Yaskawa INFORM job: DEMO_ROOF_UPPER_0625_3PAINT_49.JBI

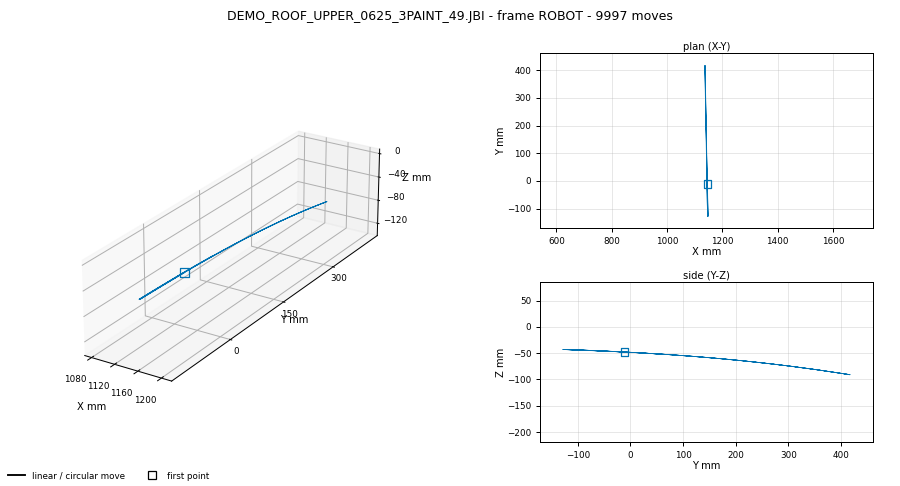
[picture p0: tool path of DEMO_ROOF_UPPER_0625_3PAINT_49.JBI in frame ROBOT, 9997 of 9997 moves have a stored position in this frame; points joined in program order, loops and branches not executed]
/JOB
//NAME DEMO_ROOF_UPPER_0625_3PAINT49
//POS
///NPOS 9997,0,0,0,0,0
///TOOL 0
///USER 0
///POSTYPE ROBOT
///RECTAN
///RCONF 1,0,0,0,0,0,0,0,0,0,0,0,0,0,0,0,0,0,0,0,0,0,0,0
C00000=1146.080,-11.263,-47.724,179.579,6.166,149.236
C00001=1146.085,-11.512,-47.711,179.577,6.165,149.237
C00002=1146.092,-11.763,-47.699,179.574,6.165,149.238
C00003=1146.097,-12.012,-47.686,179.572,6.164,149.238
C00004=1146.101,-12.262,-47.673,179.570,6.163,149.239
C00005=1146.106,-12.511,-47.661,179.567,6.163,149.239
C00006=1146.112,-12.761,-47.648,179.565,6.162,149.240
C00007=1146.117,-13.010,-47.635,179.563,6.161,149.240
C00008=1146.122,-13.261,-47.623,179.560,6.161,149.241
C00009=1146.127,-13.510,-47.610,179.558,6.160,149.242
C00010=1146.132,-13.760,-47.597,179.555,6.159,149.242
C00011=1146.138,-14.009,-47.585,179.552,6.158,149.243
C00012=1146.143,-14.258,-47.572,179.550,6.157,149.243
C00013=1146.148,-14.509,-47.560,179.548,6.156,149.244
C00014=1146.153,-14.758,-47.547,179.545,6.156,149.244
C00015=1146.158,-15.007,-47.535,179.543,6.155,149.245
C00016=1146.163,-15.257,-47.522,179.540,6.155,149.245
C00017=1146.169,-15.507,-47.510,179.538,6.154,149.246
C00018=1146.174,-15.756,-47.497,179.536,6.154,149.247
C00019=1146.179,-16.006,-47.484,179.533,6.153,149.247
C00020=1146.184,-16.256,-47.472,179.531,6.152,149.248
C00021=1146.189,-16.506,-47.460,179.529,6.152,149.248
C00022=1146.194,-16.755,-47.447,179.526,6.151,149.249
C00023=1146.200,-17.004,-47.434,179.523,6.150,149.249
C00024=1146.205,-17.254,-47.422,179.521,6.149,149.250
C00025=1146.210,-17.503,-47.410,179.518,6.148,149.251
C00026=1146.215,-17.753,-47.397,179.516,6.148,149.251
C00027=1146.220,-18.003,-47.385,179.514,6.147,149.252
C00028=1146.225,-18.253,-47.372,179.511,6.146,149.252
C00029=1146.231,-18.503,-47.361,179.509,6.146,149.253
C00030=1146.236,-18.752,-47.348,179.506,6.145,149.253
C00031=1146.241,-19.001,-47.335,179.504,6.144,149.254
C00032=1146.246,-19.251,-47.323,179.502,6.144,149.254
C00033=1146.251,-19.501,-47.311,179.499,6.143,149.255
C00034=1146.256,-19.751,-47.299,179.497,6.142,149.256
C00035=1146.261,-20.001,-47.286,179.495,6.142,149.256
C00036=1146.266,-20.250,-47.273,179.492,6.141,149.257
C00037=1146.272,-20.500,-47.262,179.490,6.141,149.257
C00038=1146.277,-20.749,-47.249,179.488,6.140,149.258
C00039=1146.282,-20.999,-47.237,179.485,6.139,149.258
C00040=1146.288,-21.248,-47.224,179.483,6.139,149.259
C00041=1146.293,-21.498,-47.213,179.481,6.138,149.259
C00042=1146.298,-21.748,-47.200,179.477,6.137,149.260
C00043=1146.304,-21.998,-47.188,179.475,6.136,149.261
C00044=1146.309,-22.247,-47.175,179.472,6.135,149.261
C00045=1146.314,-22.497,-47.164,179.470,6.135,149.262
C00046=1146.319,-22.746,-47.151,179.468,6.134,149.262
C00047=1146.325,-22.996,-47.139,179.465,6.133,149.263
C00048=1146.330,-23.245,-47.127,179.463,6.133,149.263
C00049=1146.335,-23.496,-47.114,179.461,6.132,149.264
C00050=1146.340,-23.745,-47.102,179.458,6.131,149.265
C00051=1146.345,-23.995,-47.090,179.456,6.131,149.265
C00052=1146.351,-24.264,-47.076,179.454,6.130,149.266
C00053=1146.356,-24.535,-47.063,179.451,6.130,149.266
C00054=1146.361,-24.805,-47.051,179.449,6.129,149.267
C00055=1146.367,-25.075,-47.038,179.445,6.128,149.268
C00056=1146.372,-25.324,-47.025,179.443,6.127,149.268
C00057=1146.378,-25.574,-47.013,179.441,6.127,149.269
C00058=1146.383,-25.824,-47.002,179.438,6.126,149.269
C00059=1146.388,-26.073,-46.989,179.436,6.125,149.270
C00060=1146.394,-26.323,-46.977,179.434,6.125,149.270
C00061=1146.399,-26.572,-46.964,179.431,6.124,149.271
C00062=1146.404,-26.822,-46.953,179.429,6.123,149.272
C00063=1146.409,-27.072,-46.941,179.427,6.123,149.272
C00064=1146.414,-27.321,-46.929,179.424,6.122,149.273
C00065=1146.420,-27.571,-46.917,179.422,6.121,149.273
C00066=1146.425,-27.821,-46.905,179.419,6.121,149.274
C00067=1146.429,-28.070,-46.893,179.417,6.120,149.274
C00068=1146.435,-28.320,-46.881,179.415,6.119,149.275
C00069=1146.440,-28.570,-46.869,179.412,6.119,149.276
C00070=1146.445,-28.819,-46.857,179.410,6.118,149.276
C00071=1146.451,-29.069,-46.845,179.407,6.118,149.277
C00072=1146.456,-29.319,-46.833,179.405,6.117,149.277
C00073=1146.461,-29.568,-46.821,179.402,6.117,149.278
C00074=1146.466,-29.818,-46.809,179.400,6.116,149.278
C00075=1146.472,-30.068,-46.797,179.398,6.115,149.279
C00076=1146.476,-30.318,-46.786,179.395,6.115,149.280
C00077=1146.481,-30.567,-46.773,179.393,6.114,149.280
C00078=1146.487,-30.817,-46.761,179.390,6.113,149.281
C00079=1146.492,-31.067,-46.749,179.388,6.113,149.281
C00080=1146.497,-31.317,-46.738,179.387,6.113,149.282
C00081=1146.503,-31.566,-46.727,179.384,6.112,149.282
C00082=1146.508,-31.815,-46.714,179.382,6.111,149.283
C00083=1146.513,-32.065,-46.702,179.379,6.111,149.284
C00084=1146.518,-32.315,-46.691,179.377,6.110,149.284
C00085=1146.524,-32.565,-46.679,179.374,6.110,149.285
C00086=1146.529,-32.815,-46.667,179.372,6.109,149.285
C00087=1146.533,-33.064,-46.655,179.370,6.108,149.286
C00088=1146.539,-33.313,-46.643,179.367,6.108,149.286
C00089=1146.544,-33.563,-46.631,179.365,6.107,149.287
C00090=1146.549,-33.813,-46.620,179.362,6.107,149.288
C00091=1146.555,-34.062,-46.608,179.360,6.106,149.288
C00092=1146.560,-34.312,-46.597,179.358,6.105,149.289
C00093=1146.565,-34.562,-46.585,179.355,6.105,149.289
C00094=1146.570,-34.811,-46.573,179.353,6.104,149.290
C00095=1146.576,-35.061,-46.561,179.351,6.103,149.290
C00096=1146.580,-35.311,-46.549,179.348,6.103,149.291
C00097=1146.586,-35.561,-46.538,179.346,6.102,149.291
C00098=1146.592,-35.810,-46.526,179.344,6.101,149.292
C00099=1146.596,-36.060,-46.515,179.341,6.101,149.293
C00100=1146.602,-36.309,-46.503,179.339,6.100,149.293
C00101=1146.607,-36.559,-46.492,179.336,6.099,149.294
C00102=1146.612,-36.809,-46.480,179.334,6.099,149.294
C00103=1146.617,-37.059,-46.468,179.332,6.098,149.295
C00104=1146.622,-37.309,-46.457,179.329,6.097,149.295
C00105=1146.628,-37.558,-46.445,179.327,6.097,149.296
C00106=1146.633,-37.807,-46.434,179.325,6.097,149.297
C00107=1146.638,-38.057,-46.422,179.323,6.097,149.297
C00108=1146.644,-38.307,-46.410,179.320,6.096,149.298
C00109=1146.648,-38.557,-46.399,179.318,6.095,149.298
C00110=1146.654,-38.806,-46.387,179.315,6.095,149.299
C00111=1146.659,-39.056,-46.376,179.313,6.094,149.299
C00112=1146.665,-39.306,-46.364,179.311,6.093,149.300
C00113=1146.670,-39.556,-46.352,179.308,6.093,149.301
C00114=1146.675,-39.805,-46.341,179.306,6.092,149.301
C00115=1146.681,-40.055,-46.329,179.304,6.091,149.302
C00116=1146.685,-40.304,-46.318,179.301,6.091,149.302
C00117=1146.691,-40.554,-46.306,179.299,6.090,149.303
C00118=1146.696,-40.804,-46.295,179.297,6.089,149.303
C00119=1146.701,-41.054,-46.283,179.294,6.089,149.304
C00120=1146.706,-41.303,-46.272,179.292,6.088,149.305
C00121=1146.712,-41.553,-46.260,179.290,6.088,149.305
C00122=1146.717,-41.803,-46.250,179.287,6.088,149.306
C00123=1146.722,-42.053,-46.238,179.285,6.087,149.306
C00124=1146.727,-42.302,-46.227,179.283,6.086,149.307
C00125=1146.733,-42.552,-46.215,179.280,6.086,149.307
C00126=1146.738,-42.801,-46.204,179.278,6.085,149.308
C00127=1146.743,-43.051,-46.192,179.276,6.084,149.308
C00128=1146.748,-43.300,-46.181,179.273,6.084,149.309
C00129=1146.754,-43.551,-46.170,179.271,6.083,149.310
C00130=1146.759,-43.800,-46.158,179.269,6.083,149.310
C00131=1146.763,-44.050,-46.147,179.266,6.082,149.311
C00132=1146.769,-44.299,-46.135,179.264,6.081,149.311
C00133=1146.774,-44.549,-46.124,179.262,6.082,149.312
C00134=1146.780,-44.799,-46.112,179.260,6.081,149.312
C00135=1146.785,-45.049,-46.102,179.257,6.080,149.313
C00136=1146.791,-45.298,-46.090,179.255,6.080,149.314
C00137=1146.795,-45.548,-46.079,179.253,6.079,149.314
C00138=1146.800,-45.797,-46.068,179.250,6.078,149.315
C00139=1146.806,-46.047,-46.057,179.248,6.078,149.315
C00140=1146.811,-46.297,-46.046,179.245,6.077,149.316
C00141=1146.816,-46.547,-46.034,179.243,6.076,149.316
C00142=1146.822,-46.796,-46.023,179.242,6.076,149.317
C00143=1146.827,-47.046,-46.012,179.239,6.076,149.318
C00144=1146.832,-47.296,-46.000,179.237,6.075,149.318
C00145=1146.837,-47.545,-45.989,179.234,6.075,149.319
C00146=1146.843,-47.795,-45.977,179.232,6.074,149.319
C00147=1146.848,-48.045,-45.967,179.230,6.073,149.320
C00148=1146.853,-48.294,-45.956,179.227,6.073,149.320
C00149=1146.859,-48.544,-45.944,179.225,6.072,149.321
C00150=1146.864,-48.794,-45.933,179.223,6.071,149.321
C00151=1146.869,-49.043,-45.923,179.221,6.072,149.322
C00152=1146.874,-49.293,-45.911,179.218,6.071,149.322
C00153=1146.879,-49.543,-45.900,179.216,6.071,149.323
C00154=1146.885,-49.792,-45.889,179.214,6.070,149.324
C00155=1146.890,-50.042,-45.877,179.211,6.069,149.324
C00156=1146.895,-50.313,-45.866,179.209,6.069,149.325
C00157=1146.901,-50.583,-45.854,179.206,6.068,149.326
C00158=1146.907,-50.854,-45.841,179.204,6.067,149.326
C00159=1146.912,-51.125,-45.829,179.201,6.067,149.327
C00160=1146.918,-51.375,-45.819,179.199,6.066,149.327
C00161=1146.923,-51.624,-45.808,179.197,6.065,149.328
C00162=1146.929,-51.874,-45.797,179.194,6.065,149.328
C00163=1146.934,-52.124,-45.786,179.192,6.064,149.329
C00164=1146.938,-52.373,-45.774,179.190,6.065,149.330
C00165=1146.945,-52.623,-45.764,179.188,6.064,149.330
C00166=1146.949,-52.873,-45.752,179.185,6.063,149.331
C00167=1146.954,-53.123,-45.742,179.183,6.063,149.331
C00168=1146.960,-53.372,-45.731,179.181,6.062,149.332
C00169=1146.965,-53.622,-45.720,179.178,6.061,149.332
C00170=1146.971,-53.871,-45.709,179.176,6.061,149.333
C00171=1146.976,-54.122,-45.698,179.174,6.061,149.333
C00172=1146.981,-54.371,-45.687,179.171,6.060,149.334
C00173=1146.986,-54.621,-45.677,179.169,6.060,149.335
C00174=1146.991,-54.871,-45.665,179.167,6.059,149.335
C00175=1146.997,-55.120,-45.655,179.164,6.058,149.336
C00176=1147.002,-55.370,-45.643,179.162,6.058,149.336
C00177=1147.007,-55.619,-45.633,179.161,6.058,149.337
C00178=1147.012,-55.869,-45.622,179.158,6.057,149.337
C00179=1147.018,-56.120,-45.611,179.156,6.057,149.338
C00180=1147.023,-56.369,-45.600,179.154,6.056,149.338
C00181=1147.028,-56.619,-45.589,179.151,6.055,149.339
C00182=1147.033,-56.868,-45.578,179.149,6.055,149.340
C00183=1147.038,-57.118,-45.568,179.146,6.054,149.340
C00184=1147.044,-57.368,-45.557,179.144,6.054,149.341
C00185=1147.049,-57.617,-45.546,179.142,6.053,149.341
C00186=1147.055,-57.867,-45.535,179.140,6.053,149.342
C00187=1147.060,-58.117,-45.524,179.137,6.052,149.342
C00188=1147.065,-58.366,-45.514,179.135,6.051,149.343
C00189=1147.070,-58.616,-45.503,179.133,6.052,149.344
C00190=1147.076,-58.865,-45.492,179.131,6.051,149.344
C00191=1147.081,-59.116,-45.482,179.129,6.050,149.345
C00192=1147.085,-59.365,-45.470,179.126,6.050,149.345
C00193=1147.091,-59.615,-45.460,179.124,6.049,149.346
C00194=1147.097,-59.865,-45.449,179.121,6.049,149.346
C00195=1147.102,-60.114,-45.438,179.120,6.049,149.347
C00196=1147.107,-60.364,-45.428,179.118,6.048,149.347
C00197=1147.112,-60.614,-45.417,179.115,6.048,149.348
C00198=1147.117,-60.864,-45.406,179.113,6.047,149.349
C00199=1147.123,-61.113,-45.396,179.110,6.046,149.349
C00200=1147.128,-61.363,-45.385,179.108,6.046,149.350
C00201=1147.133,-61.613,-45.375,179.106,6.046,149.350
C00202=1147.139,-61.862,-45.364,179.104,6.045,149.351
C00203=1147.144,-62.112,-45.354,179.101,6.045,149.351
C00204=1147.149,-62.362,-45.343,179.099,6.044,149.352
C00205=1147.154,-62.611,-45.332,179.097,6.043,149.352
C00206=1147.159,-62.861,-45.322,179.095,6.043,149.353
C00207=1147.164,-63.111,-45.311,179.093,6.043,149.354
C00208=1147.170,-63.361,-45.301,179.091,6.042,149.354
C00209=1147.175,-63.610,-45.290,179.088,6.041,149.355
C00210=1147.180,-63.860,-45.280,179.086,6.041,149.355
C00211=1147.186,-64.110,-45.268,179.084,6.041,149.356
C00212=1147.192,-64.360,-45.258,179.081,6.040,149.356
C00213=1147.197,-64.610,-45.248,179.079,6.040,149.357
C00214=1147.202,-64.859,-45.237,179.077,6.039,149.358
C00215=1147.208,-65.109,-45.226,179.074,6.038,149.358
C00216=1147.213,-65.359,-45.216,179.073,6.038,149.359
C00217=1147.218,-65.608,-45.206,179.070,6.038,149.359
C00218=1147.222,-65.858,-45.196,179.068,6.037,149.360
C00219=1147.228,-66.107,-45.185,179.066,6.036,149.360
C00220=1147.233,-66.357,-45.175,179.064,6.037,149.361
C00221=1147.238,-66.607,-45.164,179.061,6.036,149.361
C00222=1147.244,-66.857,-45.154,179.059,6.035,149.362
C00223=1147.249,-67.107,-45.143,179.057,6.035,149.363
C00224=1147.255,-67.356,-45.133,179.054,6.034,149.363
C00225=1147.260,-67.606,-45.123,179.053,6.034,149.364
C00226=1147.265,-67.856,-45.111,179.050,6.034,149.364
C00227=1147.270,-68.105,-45.101,179.048,6.033,149.365
C00228=1147.275,-68.355,-45.091,179.046,6.032,149.365
C00229=1147.281,-68.605,-45.080,179.044,6.033,149.366
C00230=1147.287,-68.854,-45.070,179.041,6.032,149.366
C00231=1147.292,-69.105,-45.060,179.039,6.031,149.367
C00232=1147.297,-69.354,-45.049,179.037,6.031,149.368
C00233=1147.303,-69.604,-45.039,179.034,6.030,149.368
C00234=1147.308,-69.854,-45.029,179.033,6.030,149.369
C00235=1147.313,-70.103,-45.019,179.030,6.030,149.369
C00236=1147.318,-70.353,-45.009,179.028,6.029,149.370
C00237=1147.323,-70.603,-44.998,179.026,6.028,149.370
C00238=1147.329,-70.853,-44.988,179.024,6.028,149.371
C00239=1147.334,-71.103,-44.978,179.022,6.028,149.371
C00240=1147.339,-71.352,-44.967,179.019,6.027,149.372
C00241=1147.345,-71.602,-44.957,179.017,6.026,149.372
C00242=1147.350,-71.852,-44.947,179.015,6.027,149.373
C00243=1147.355,-72.101,-44.937,179.013,6.026,149.374
C00244=1147.361,-72.351,-44.927,179.011,6.025,149.374
C00245=1147.366,-72.601,-44.916,179.008,6.025,149.375
C00246=1147.371,-72.851,-44.906,179.006,6.025,149.375
C00247=1147.377,-73.100,-44.896,179.004,6.024,149.376
C00248=1147.382,-73.350,-44.886,179.002,6.024,149.376
C00249=1147.387,-73.600,-44.875,178.999,6.023,149.377
C00250=1147.392,-73.849,-44.865,178.998,6.023,149.377
C00251=1147.398,-74.099,-44.855,178.995,6.022,149.378
C00252=1147.403,-74.349,-44.845,178.993,6.022,149.379
C00253=1147.408,-74.599,-44.834,178.991,6.021,149.379
C00254=1147.414,-74.848,-44.824,178.989,6.021,149.380
C00255=1147.418,-75.098,-44.814,178.986,6.020,149.380
C00256=1147.424,-75.348,-44.804,178.984,6.020,149.381
C00257=1147.429,-75.597,-44.794,178.982,6.019,149.381
C00258=1147.435,-75.847,-44.784,178.980,6.019,149.382
C00259=1147.440,-76.098,-44.774,178.978,6.019,149.382
C00260=1147.446,-76.368,-44.763,178.975,6.018,149.383
C00261=1147.451,-76.639,-44.752,178.973,6.017,149.384
C00262=1147.457,-76.911,-44.741,178.970,6.017,149.384
C00263=1147.463,-77.182,-44.731,178.968,6.016,149.385
C00264=1147.468,-77.433,-44.720,178.966,6.016,149.385
C00265=1147.474,-77.682,-44.710,178.964,6.016,149.386
C00266=1147.480,-77.932,-44.700,178.962,6.015,149.387
C00267=1147.484,-78.181,-44.690,178.959,6.014,149.387
C00268=1147.490,-78.432,-44.680,178.957,6.015,149.388
C00269=1147.495,-78.681,-44.670,178.955,6.014,149.388
C00270=1147.501,-78.931,-44.660,178.953,6.013,149.389
C00271=1147.506,-79.180,-44.650,178.951,6.013,149.389
C00272=1147.511,-79.430,-44.640,178.949,6.013,149.390
C00273=1147.517,-79.680,-44.630,178.946,6.012,149.390
C00274=1147.521,-79.930,-44.621,178.944,6.011,149.391
C00275=1147.527,-80.179,-44.610,178.942,6.012,149.392
C00276=1147.533,-80.429,-44.600,178.940,6.011,149.392
C00277=1147.537,-80.679,-44.591,178.938,6.010,149.392
C00278=1147.543,-80.929,-44.581,178.936,6.011,149.393
C00279=1147.548,-81.178,-44.570,178.934,6.010,149.394
C00280=1147.553,-81.428,-44.561,178.931,6.009,149.394
C00281=1147.559,-81.678,-44.551,178.929,6.008,149.395
C00282=1147.564,-81.928,-44.541,178.927,6.009,149.395
C00283=1147.569,-82.177,-44.531,178.925,6.008,149.396
C00284=1147.575,-82.427,-44.521,178.923,6.007,149.396
C00285=1147.581,-82.677,-44.511,178.921,6.008,149.397
C00286=1147.585,-82.926,-44.502,178.918,6.007,149.398
C00287=1147.590,-83.176,-44.491,178.916,6.006,149.398
C00288=1147.596,-83.427,-44.482,178.914,6.005,149.398
C00289=1147.601,-83.676,-44.472,178.912,6.006,149.399
C00290=1147.607,-83.925,-44.462,178.910,6.005,149.400
C00291=1147.612,-84.175,-44.453,178.908,6.004,149.400
C00292=1147.618,-84.425,-44.443,178.906,6.004,149.401
C00293=1147.623,-84.675,-44.432,178.903,6.004,149.401
C00294=1147.628,-84.925,-44.423,178.901,6.003,149.402
C00295=1147.633,-85.174,-44.413,178.900,6.003,149.402
C00296=1147.638,-85.424,-44.404,178.897,6.003,149.403
C00297=1147.644,-85.674,-44.394,178.895,6.002,149.404
C00298=1147.650,-85.923,-44.384,178.893,6.002,149.404
C00299=1147.655,-86.173,-44.375,178.891,6.001,149.404
C00300=1147.660,-86.423,-44.364,178.888,6.001,149.405
C00301=1147.665,-86.673,-44.356,178.886,6.000,149.406
C00302=1147.671,-86.923,-44.345,178.884,6.000,149.406
C00303=1147.675,-87.172,-44.336,178.882,5.999,149.407
C00304=1147.681,-87.422,-44.326,178.880,5.999,149.407
C00305=1147.686,-87.671,-44.317,178.878,5.999,149.408
C00306=1147.692,-87.922,-44.307,178.876,5.998,149.408
C00307=1147.697,-88.171,-44.297,178.873,5.998,149.409
C00308=1147.702,-88.422,-44.288,178.872,5.998,149.410
C00309=1147.707,-88.671,-44.278,178.869,5.997,149.410
C00310=1147.713,-88.921,-44.269,178.867,5.996,149.410
C00311=1147.718,-89.170,-44.259,178.865,5.997,149.411
C00312=1147.724,-89.421,-44.249,178.863,5.996,149.412
C00313=1147.729,-89.670,-44.240,178.861,5.995,149.412
C00314=1147.735,-89.920,-44.230,178.859,5.995,149.413
C00315=1147.739,-90.169,-44.221,178.856,5.995,149.413
C00316=1147.745,-90.419,-44.211,178.854,5.994,149.414
C00317=1147.750,-90.669,-44.202,178.853,5.994,149.414
C00318=1147.756,-90.919,-44.192,178.850,5.994,149.415
C00319=1147.760,-91.169,-44.182,178.848,5.993,149.416
C00320=1147.766,-91.419,-44.173,178.846,5.993,149.416
C00321=1147.771,-91.668,-44.163,178.844,5.992,149.416
C00322=1147.777,-91.918,-44.154,178.842,5.992,149.417
C00323=1147.782,-92.167,-44.144,178.840,5.992,149.418
C00324=1147.788,-92.418,-44.134,178.837,5.991,149.418
C00325=1147.793,-92.667,-44.125,178.835,5.991,149.419
C00326=1147.798,-92.917,-44.116,178.834,5.991,149.419
C00327=1147.804,-93.167,-44.106,178.831,5.990,149.420
C00328=1147.809,-93.416,-44.097,178.829,5.989,149.420
C00329=1147.815,-93.666,-44.087,178.827,5.989,149.421
C00330=1147.819,-93.915,-44.078,178.825,5.989,149.421
C00331=1147.825,-94.166,-44.068,178.823,5.989,149.422
C00332=1147.830,-94.415,-44.059,178.821,5.988,149.422
C00333=1147.835,-94.665,-44.050,178.819,5.988,149.423
C00334=1147.841,-94.915,-44.040,178.817,5.988,149.423
C00335=1147.846,-95.165,-44.031,178.815,5.987,149.424
C00336=1147.852,-95.414,-44.021,178.812,5.987,149.425
C00337=1147.857,-95.664,-44.012,178.811,5.987,149.425
C00338=1147.862,-95.914,-44.003,178.808,5.986,149.426
C00339=1147.868,-96.164,-43.993,178.806,5.985,149.426
C00340=1147.873,-96.413,-43.984,178.804,5.985,149.427
C00341=1147.878,-96.663,-43.975,178.802,5.985,149.427
C00342=1147.884,-96.913,-43.965,178.800,5.984,149.428
C00343=1147.889,-97.163,-43.956,178.798,5.984,149.428
C00344=1147.895,-97.413,-43.947,178.796,5.983,149.429
C00345=1147.900,-97.662,-43.937,178.794,5.984,149.429
C00346=1147.905,-97.912,-43.928,178.792,5.983,149.430
C00347=1147.911,-98.162,-43.919,178.789,5.982,149.430
C00348=1147.916,-98.412,-43.910,178.788,5.982,149.431
C00349=1147.921,-98.661,-43.900,178.785,5.982,149.432
C00350=1147.927,-98.911,-43.891,178.783,5.981,149.432
C00351=1147.932,-99.161,-43.882,178.781,5.981,149.433
C00352=1147.937,-99.411,-43.873,178.779,5.980,149.433
C00353=1147.943,-99.661,-43.863,178.778,5.980,149.434
C00354=1147.948,-99.910,-43.854,178.775,5.980,149.434
C00355=1147.953,-100.160,-43.845,178.773,5.979,149.435
C00356=1147.958,-100.410,-43.836,178.771,5.979,149.435
C00357=1147.964,-100.660,-43.826,178.769,5.979,149.436
C00358=1147.969,-100.909,-43.817,178.767,5.979,149.436
C00359=1147.974,-101.159,-43.808,178.765,5.978,149.437
C00360=1147.980,-101.409,-43.798,178.762,5.977,149.437
C00361=1147.985,-101.659,-43.790,178.761,5.977,149.438
C00362=1147.991,-101.908,-43.781,178.759,5.977,149.438
C00363=1147.996,-102.158,-43.771,178.756,5.976,149.439
C00364=1148.002,-102.430,-43.762,178.754,5.976,149.440
C00365=1148.008,-102.702,-43.751,178.752,5.976,149.440
C00366=1148.014,-102.975,-43.742,178.749,5.975,149.441
C00367=1148.019,-103.247,-43.731,178.747,5.975,149.441
C00368=1148.024,-103.497,-43.722,178.746,5.975,149.442
C00369=1148.030,-103.747,-43.714,178.743,5.974,149.442
C00370=1148.036,-103.996,-43.704,178.741,5.974,149.443
C00371=1148.041,-104.246,-43.696,178.739,5.973,149.443
C00372=1148.046,-104.495,-43.686,178.737,5.973,149.444
C00373=1148.051,-104.745,-43.677,178.735,5.973,149.444
C00374=1148.056,-104.995,-43.668,178.733,5.972,149.445
C00375=1148.062,-105.245,-43.659,178.731,5.972,149.446
C00376=1148.067,-105.495,-43.650,178.729,5.972,149.446
C00377=1148.073,-105.745,-43.641,178.727,5.971,149.447
C00378=1148.078,-105.995,-43.632,178.725,5.971,149.447
C00379=1148.084,-106.244,-43.623,178.723,5.970,149.448
C00380=1148.089,-106.494,-43.615,178.721,5.970,149.448
C00381=1148.095,-106.744,-43.605,178.719,5.970,149.449
C00382=1148.100,-106.994,-43.596,178.716,5.969,149.449
C00383=1148.105,-107.243,-43.587,178.715,5.969,149.450
C00384=1148.110,-107.493,-43.578,178.713,5.968,149.450
C00385=1148.115,-107.743,-43.569,178.711,5.968,149.451
C00386=1148.120,-107.993,-43.561,178.709,5.968,149.451
C00387=1148.127,-108.243,-43.551,178.707,5.968,149.452
C00388=1148.132,-108.492,-43.542,178.705,5.967,149.452
C00389=1148.137,-108.742,-43.534,178.702,5.967,149.453
C00390=1148.142,-108.992,-43.525,178.701,5.967,149.453
C00391=1148.148,-109.242,-43.516,178.699,5.966,149.454
C00392=1148.153,-109.492,-43.507,178.697,5.966,149.454
C00393=1148.159,-109.741,-43.498,178.694,5.966,149.455
C00394=1148.164,-109.991,-43.489,178.693,5.966,149.456
C00395=1148.169,-110.241,-43.481,178.691,5.965,149.456
C00396=1148.175,-110.491,-43.471,178.688,5.964,149.457
C00397=1148.180,-110.741,-43.462,178.687,5.964,149.457
C00398=1148.185,-110.990,-43.453,178.685,5.963,149.458
C00399=1148.191,-111.240,-43.445,178.683,5.964,149.458
C00400=1148.196,-111.489,-43.436,178.680,5.963,149.459
C00401=1148.201,-111.739,-43.427,178.679,5.963,149.459
C00402=1148.206,-111.989,-43.418,178.677,5.962,149.460
C00403=1148.212,-112.239,-43.409,178.674,5.962,149.460
C00404=1148.217,-112.488,-43.401,178.673,5.962,149.461
C00405=1148.222,-112.738,-43.392,178.671,5.961,149.461
C00406=1148.228,-112.989,-43.384,178.668,5.961,149.462
C00407=1148.233,-113.238,-43.375,178.666,5.961,149.462
C00408=1148.239,-113.487,-43.366,178.665,5.961,149.463
C00409=1148.245,-113.738,-43.357,178.662,5.960,149.463
C00410=1148.250,-113.988,-43.348,178.660,5.959,149.464
C00411=1148.255,-114.237,-43.339,178.659,5.959,149.464
C00412=1148.260,-114.487,-43.330,178.656,5.958,149.465
C00413=1148.266,-114.737,-43.322,178.654,5.959,149.465
C00414=1148.272,-114.987,-43.313,178.652,5.958,149.466
C00415=1148.277,-115.237,-43.304,178.651,5.958,149.466
C00416=1148.282,-115.487,-43.295,178.648,5.957,149.467
C00417=1148.288,-115.736,-43.287,178.647,5.957,149.467
C00418=1148.293,-115.986,-43.278,178.645,5.957,149.468
C00419=1148.298,-116.236,-43.270,178.642,5.956,149.468
C00420=1148.303,-116.486,-43.261,178.640,5.956,149.469
C00421=1148.309,-116.735,-43.252,178.638,5.956,149.470
C00422=1148.314,-116.985,-43.243,178.637,5.956,149.470
C00423=1148.320,-117.235,-43.235,178.634,5.955,149.471
C00424=1148.326,-117.484,-43.227,178.633,5.955,149.471
C00425=1148.331,-117.734,-43.218,178.631,5.954,149.472
C00426=1148.336,-117.984,-43.209,178.629,5.954,149.472
C00427=1148.341,-118.234,-43.200,178.627,5.953,149.473
C00428=1148.347,-118.484,-43.192,178.625,5.954,149.473
C00429=1148.352,-118.733,-43.184,178.623,5.953,149.474
C00430=1148.357,-118.983,-43.175,178.621,5.953,149.474
C00431=1148.362,-119.233,-43.166,178.619,5.952,149.475
C00432=1148.368,-119.483,-43.158,178.617,5.952,149.475
C00433=1148.373,-119.733,-43.149,178.615,5.952,149.476
C00434=1148.378,-119.983,-43.141,178.613,5.951,149.476
C00435=1148.384,-120.232,-43.133,178.611,5.951,149.477
C00436=1148.390,-120.482,-43.124,178.609,5.950,149.477
C00437=1148.395,-120.732,-43.115,178.607,5.951,149.478
C00438=1148.401,-120.981,-43.106,178.605,5.950,149.478
C00439=1148.406,-121.232,-43.098,178.603,5.950,149.479
C00440=1148.411,-121.481,-43.089,178.601,5.949,149.479
C00441=1148.416,-121.730,-43.081,178.599,5.949,149.480
C00442=1148.422,-121.981,-43.073,178.597,5.948,149.480
C00443=1148.427,-122.231,-43.064,178.595,5.948,149.481
C00444=1148.432,-122.480,-43.055,178.593,5.948,149.481
C00445=1148.438,-122.730,-43.048,178.592,5.948,149.482
C00446=1148.443,-122.980,-43.039,178.589,5.947,149.482
C00447=1148.449,-123.229,-43.030,178.588,5.947,149.483
C00448=1148.454,-123.480,-43.022,178.585,5.947,149.483
C00449=1148.459,-123.729,-43.014,178.584,5.947,149.484
C00450=1148.465,-123.979,-43.006,178.581,5.946,149.484
C00451=1148.470,-124.229,-42.997,178.579,5.945,149.485
C00452=1148.475,-124.479,-42.988,178.578,5.945,149.485
C00453=1148.481,-124.728,-42.980,178.575,5.945,149.486
C00454=1148.487,-124.978,-42.971,178.574,5.945,149.486
C00455=1148.492,-125.229,-42.963,178.572,5.944,149.487
C00456=1148.497,-125.478,-42.955,178.570,5.944,149.487
C00457=1148.502,-125.728,-42.946,178.568,5.943,149.488
C00458=1148.508,-125.978,-42.938,178.566,5.943,149.488
C00459=1148.513,-126.227,-42.930,178.564,5.942,149.489
C00460=1148.519,-126.478,-42.921,178.562,5.943,149.490
C00461=1148.524,-126.726,-42.913,178.560,5.942,149.490
C00462=1148.529,-126.977,-42.905,178.558,5.942,149.491
C00463=1148.535,-127.227,-42.896,178.556,5.941,149.491
C00464=1148.541,-127.477,-42.889,178.554,5.941,149.491
C00465=1148.546,-127.726,-42.880,178.552,5.941,149.492
C00466=1148.551,-127.976,-42.872,178.551,5.941,149.492
C00467=1148.556,-128.226,-42.864,178.548,5.940,149.493
C00468=1148.135,-128.237,-42.906,178.545,5.944,149.495
C00469=1148.130,-127.987,-42.915,178.547,5.944,149.494
C00470=1148.124,-127.737,-42.923,178.549,5.945,149.494
C00471=1148.119,-127.488,-42.931,178.551,5.945,149.493
C00472=1148.114,-127.238,-42.939,178.553,5.945,149.493
C00473=1148.108,-126.988,-42.948,178.555,5.945,149.492
C00474=1148.103,-126.738,-42.956,178.557,5.946,149.492
C00475=1148.098,-126.488,-42.965,178.559,5.946,149.491
C00476=1148.092,-126.239,-42.972,178.561,5.947,149.491
C00477=1148.087,-125.989,-42.981,178.562,5.946,149.490
C00478=1148.082,-125.739,-42.990,178.565,5.947,149.490
C00479=1148.076,-125.489,-42.998,178.566,5.947,149.489
C00480=1148.071,-125.239,-43.007,178.568,5.948,149.489
C00481=1148.065,-124.990,-43.014,178.570,5.948,149.488
C00482=1148.060,-124.740,-43.023,178.572,5.949,149.488
C00483=1148.055,-124.490,-43.031,178.574,5.949,149.487
C00484=1148.049,-124.240,-43.039,178.576,5.949,149.487
C00485=1148.044,-123.991,-43.048,178.578,5.949,149.486
C00486=1148.038,-123.740,-43.056,178.580,5.950,149.486
C00487=1148.032,-123.491,-43.065,178.582,5.950,149.485
C00488=1148.028,-123.241,-43.073,178.584,5.950,149.485
C00489=1148.023,-122.991,-43.082,178.586,5.951,149.484
C00490=1148.017,-122.742,-43.090,178.588,5.951,149.484
C00491=1148.011,-122.491,-43.098,178.590,5.952,149.483
C00492=1148.006,-122.241,-43.107,178.592,5.952,149.483
C00493=1148.000,-121.992,-43.116,178.594,5.953,149.482
C00494=1147.995,-121.742,-43.124,178.595,5.952,149.482
C00495=1147.990,-121.492,-43.133,178.598,5.953,149.481
C00496=1147.985,-121.243,-43.141,178.599,5.953,149.481
C00497=1147.979,-120.993,-43.149,178.602,5.954,149.480
C00498=1147.974,-120.743,-43.158,178.603,5.953,149.479
C00499=1147.968,-120.494,-43.166,178.606,5.954,149.479
C00500=1147.963,-120.244,-43.175,178.607,5.954,149.478
C00501=1147.958,-119.993,-43.183,178.609,5.955,149.478
C00502=1147.953,-119.743,-43.192,178.611,5.955,149.478
C00503=1147.947,-119.494,-43.201,178.613,5.956,149.477
C00504=1147.941,-119.244,-43.209,178.615,5.956,149.477
C00505=1147.936,-118.994,-43.218,178.617,5.956,149.476
C00506=1147.930,-118.745,-43.226,178.619,5.957,149.476
C00507=1147.925,-118.495,-43.235,178.621,5.957,149.475
C00508=1147.920,-118.245,-43.243,178.624,5.957,149.474
C00509=1147.915,-117.995,-43.252,178.625,5.957,149.474
C00510=1147.910,-117.746,-43.260,178.627,5.958,149.473
C00511=1147.904,-117.496,-43.269,178.629,5.958,149.473
C00512=1147.899,-117.246,-43.277,178.631,5.959,149.472
C00513=1147.893,-116.996,-43.286,178.633,5.959,149.472
C00514=1147.888,-116.747,-43.295,178.635,5.960,149.471
C00515=1147.883,-116.497,-43.304,178.637,5.959,149.471
C00516=1147.878,-116.247,-43.313,178.639,5.960,149.470
C00517=1147.872,-115.997,-43.320,178.641,5.960,149.470
C00518=1147.866,-115.747,-43.329,178.643,5.961,149.469
C00519=1147.861,-115.497,-43.338,178.645,5.961,149.469
C00520=1147.856,-115.247,-43.347,178.647,5.961,149.468
C00521=1147.850,-114.998,-43.356,178.649,5.962,149.468
C00522=1147.845,-114.748,-43.364,178.651,5.962,149.467
C00523=1147.840,-114.498,-43.373,178.653,5.962,149.467
C00524=1147.834,-114.248,-43.382,178.655,5.962,149.466
C00525=1147.829,-113.999,-43.390,178.657,5.963,149.466
C00526=1147.824,-113.749,-43.399,178.659,5.963,149.465
C00527=1147.818,-113.499,-43.409,178.661,5.964,149.465
C00528=1147.812,-113.249,-43.417,178.663,5.965,149.464
C00529=1147.807,-112.999,-43.426,178.665,5.965,149.464
C00530=1147.801,-112.750,-43.434,178.667,5.965,149.463
C00531=1147.796,-112.500,-43.443,178.669,5.965,149.462
C00532=1147.791,-112.250,-43.452,178.671,5.966,149.462
C00533=1147.786,-112.000,-43.461,178.673,5.966,149.462
C00534=1147.780,-111.751,-43.469,178.675,5.966,149.461
C00535=1147.775,-111.501,-43.478,178.677,5.967,149.461
C00536=1147.770,-111.251,-43.487,178.679,5.967,149.460
C00537=1147.764,-111.001,-43.496,178.681,5.967,149.459
C00538=1147.759,-110.751,-43.505,178.683,5.967,149.459
C00539=1147.754,-110.502,-43.514,178.685,5.968,149.458
C00540=1147.748,-110.252,-43.522,178.687,5.968,149.458
C00541=1147.742,-110.002,-43.531,178.689,5.969,149.457
C00542=1147.737,-109.752,-43.540,178.691,5.970,149.457
C00543=1147.732,-109.502,-43.549,178.693,5.970,149.456
C00544=1147.727,-109.252,-43.558,178.695,5.970,149.456
C00545=1147.721,-109.003,-43.566,178.697,5.970,149.455
C00546=1147.716,-108.753,-43.575,178.699,5.971,149.455
C00547=1147.711,-108.503,-43.584,178.701,5.971,149.454
C00548=1147.705,-108.253,-43.593,178.703,5.971,149.454
C00549=1147.699,-108.003,-43.603,178.705,5.972,149.453
C00550=1147.694,-107.753,-43.612,178.707,5.972,149.453
C00551=1147.689,-107.504,-43.620,178.709,5.972,149.452
C00552=1147.683,-107.254,-43.629,178.711,5.972,149.452
C00553=1147.678,-107.005,-43.638,178.713,5.973,149.451
C00554=1147.673,-106.755,-43.647,178.715,5.974,149.451
C00555=1147.668,-106.505,-43.656,178.717,5.974,149.450
C00556=1147.662,-106.255,-43.666,178.720,5.974,149.449
C00557=1147.657,-106.005,-43.675,178.721,5.974,149.449
C00558=1147.652,-105.756,-43.684,178.724,5.975,149.448
C00559=1147.646,-105.506,-43.692,178.726,5.976,149.448
C00560=1147.641,-105.257,-43.701,178.727,5.976,149.447
C00561=1147.635,-105.006,-43.711,178.730,5.976,149.447
C00562=1147.630,-104.757,-43.719,178.732,5.976,149.446
C00563=1147.625,-104.507,-43.728,178.734,5.977,149.446
C00564=1147.620,-104.257,-43.737,178.735,5.977,149.445
C00565=1147.614,-104.007,-43.746,178.738,5.977,149.445
C00566=1147.609,-103.757,-43.756,178.740,5.978,149.444
C00567=1147.604,-103.508,-43.765,178.742,5.978,149.444
C00568=1147.599,-103.258,-43.774,178.744,5.979,149.443
C00569=1147.592,-102.986,-43.783,178.746,5.979,149.443
C00570=1147.587,-102.714,-43.794,178.748,5.979,149.442
C00571=1147.581,-102.441,-43.803,178.751,5.980,149.441
C00572=1147.575,-102.169,-43.814,178.753,5.980,149.441
C00573=1147.569,-101.919,-43.823,178.755,5.981,149.440
C00574=1147.564,-101.670,-43.832,178.757,5.981,149.440
C00575=1147.559,-101.420,-43.841,178.759,5.981,149.439
C00576=1147.554,-101.170,-43.851,178.761,5.981,149.439
C00577=1147.548,-100.920,-43.860,178.763,5.982,149.438
C00578=1147.543,-100.670,-43.869,178.766,5.983,149.438
C00579=1147.537,-100.421,-43.877,178.767,5.983,149.437
C00580=1147.532,-100.172,-43.887,178.769,5.983,149.437
C00581=1147.527,-99.922,-43.896,178.771,5.983,149.436
C00582=1147.521,-99.672,-43.905,178.773,5.984,149.436
C00583=1147.516,-99.422,-43.915,178.776,5.984,149.435
C00584=1147.510,-99.172,-43.923,178.777,5.984,149.434
C00585=1147.506,-98.923,-43.933,178.780,5.985,149.434
C00586=1147.500,-98.673,-43.943,178.782,5.986,149.433
C00587=1147.494,-98.423,-43.952,178.783,5.986,149.433
C00588=1147.490,-98.174,-43.961,178.786,5.986,149.432
C00589=1147.484,-97.923,-43.971,178.788,5.986,149.432
C00590=1147.479,-97.674,-43.980,178.790,5.987,149.431
C00591=1147.473,-97.424,-43.988,178.792,5.988,149.431
C00592=1147.468,-97.174,-43.999,178.794,5.987,149.430
C00593=1147.463,-96.924,-44.008,178.796,5.988,149.430
C00594=1147.457,-96.674,-44.016,178.799,5.989,149.429
C00595=1147.452,-96.425,-44.027,178.800,5.989,149.429
C00596=1147.447,-96.175,-44.036,178.802,5.989,149.428
C00597=1147.442,-95.925,-44.044,178.805,5.990,149.427
C00598=1147.436,-95.676,-44.055,178.807,5.990,149.427
C00599=1147.431,-95.426,-44.064,178.809,5.991,149.426
C00600=1147.425,-95.176,-44.073,178.810,5.991,149.426
C00601=1147.420,-94.926,-44.083,178.813,5.991,149.425
C00602=1147.415,-94.677,-44.092,178.815,5.992,149.425
C00603=1147.409,-94.426,-44.101,178.817,5.992,149.424
C00604=1147.404,-94.177,-44.111,178.819,5.992,149.424
C00605=1147.398,-93.927,-44.120,178.821,5.993,149.423
C00606=1147.393,-93.677,-44.129,178.823,5.993,149.423
C00607=1147.388,-93.428,-44.139,178.826,5.993,149.422
C00608=1147.382,-93.178,-44.148,178.828,5.994,149.422
C00609=1147.377,-92.929,-44.158,178.829,5.994,149.421
C00610=1147.371,-92.678,-44.167,178.832,5.995,149.420
C00611=1147.366,-92.428,-44.176,178.834,5.995,149.420
C00612=1147.361,-92.179,-44.186,178.836,5.995,149.420
C00613=1147.356,-91.929,-44.195,178.838,5.996,149.419
C00614=1147.350,-91.680,-44.205,178.841,5.996,149.418
C00615=1147.345,-91.429,-44.215,178.842,5.996,149.418
C00616=1147.340,-91.180,-44.224,178.844,5.997,149.417
C00617=1147.335,-90.930,-44.234,178.847,5.998,149.417
C00618=1147.330,-90.680,-44.243,178.849,5.998,149.416
C00619=1147.324,-90.430,-44.253,178.851,5.998,149.416
C00620=1147.319,-90.180,-44.262,178.853,5.999,149.415
C00621=1147.313,-89.931,-44.272,178.855,5.999,149.415
C00622=1147.308,-89.681,-44.281,178.857,5.999,149.414
C00623=1147.302,-89.431,-44.291,178.860,6.000,149.413
C00624=1147.297,-89.182,-44.300,178.861,6.000,149.413
C00625=1147.292,-88.932,-44.310,178.863,6.001,149.413
C00626=1147.287,-88.683,-44.320,178.866,6.001,149.412
C00627=1147.281,-88.432,-44.330,178.868,6.001,149.411
C00628=1147.277,-88.183,-44.339,178.870,6.002,149.411
C00629=1147.271,-87.933,-44.349,178.872,6.003,149.410
C00630=1147.266,-87.683,-44.358,178.874,6.002,149.410
C00631=1147.260,-87.433,-44.368,178.876,6.003,149.409
C00632=1147.255,-87.184,-44.378,178.879,6.004,149.409
C00633=1147.249,-86.934,-44.387,178.880,6.004,149.408
C00634=1147.243,-86.684,-44.397,178.883,6.004,149.407
C00635=1147.239,-86.434,-44.407,178.885,6.005,149.407
C00636=1147.233,-86.184,-44.417,178.887,6.005,149.407
C00637=1147.228,-85.935,-44.426,178.889,6.006,149.406
C00638=1147.223,-85.685,-44.436,178.891,6.006,149.405
C00639=1147.218,-85.435,-44.445,178.893,6.006,149.405
C00640=1147.212,-85.186,-44.456,178.895,6.007,149.404
C00641=1147.207,-84.936,-44.465,178.897,6.008,149.404
C00642=1147.202,-84.686,-44.475,178.900,6.008,149.403
C00643=1147.196,-84.436,-44.485,178.902,6.008,149.403
C00644=1147.191,-84.186,-44.494,178.904,6.009,149.402
C00645=1147.186,-83.937,-44.504,178.907,6.009,149.401
C00646=1147.180,-83.687,-44.513,178.908,6.009,149.401
C00647=1147.175,-83.438,-44.524,178.910,6.010,149.401
C00648=1147.170,-83.187,-44.534,178.913,6.011,149.400
C00649=1147.165,-82.937,-44.543,178.915,6.010,149.399
C00650=1147.159,-82.688,-44.553,178.917,6.011,149.399
C00651=1147.153,-82.438,-44.563,178.919,6.012,149.398
C00652=1147.148,-82.188,-44.572,178.921,6.012,149.398
C00653=1147.143,-81.938,-44.583,178.923,6.012,149.397
C00654=1147.138,-81.689,-44.593,178.925,6.013,149.397
C00655=1147.133,-81.439,-44.603,178.928,6.014,149.396
C00656=1147.127,-81.189,-44.612,178.930,6.013,149.396
C00657=1147.122,-80.940,-44.622,178.932,6.014,149.395
C00658=1147.117,-80.690,-44.632,178.934,6.015,149.395
C00659=1147.111,-80.440,-44.643,178.936,6.015,149.394
C00660=1147.106,-80.190,-44.652,178.938,6.015,149.393
C00661=1147.101,-79.941,-44.662,178.941,6.016,149.393
C00662=1147.095,-79.691,-44.672,178.943,6.017,149.392
C00663=1147.090,-79.441,-44.683,178.945,6.016,149.392
C00664=1147.085,-79.191,-44.691,178.947,6.017,149.391
C00665=1147.079,-78.942,-44.702,178.949,6.018,149.391
C00666=1147.074,-78.692,-44.712,178.951,6.018,149.390
C00667=1147.069,-78.443,-44.721,178.953,6.018,149.390
C00668=1147.064,-78.193,-44.732,178.956,6.019,149.389
C00669=1147.058,-77.943,-44.742,178.958,6.020,149.389
C00670=1147.052,-77.693,-44.752,178.960,6.019,149.388
C00671=1147.048,-77.444,-44.761,178.962,6.020,149.387
C00672=1147.043,-77.193,-44.772,178.964,6.021,149.387
C00673=1147.036,-76.923,-44.783,178.967,6.021,149.386
C00674=1147.030,-76.651,-44.793,178.969,6.022,149.386
C00675=1147.025,-76.379,-44.805,178.972,6.022,149.385
C00676=1147.019,-76.108,-44.815,178.973,6.022,149.384
C00677=1147.014,-75.858,-44.826,178.976,6.023,149.384
C00678=1147.008,-75.609,-44.836,178.978,6.023,149.383
C00679=1147.003,-75.359,-44.846,178.981,6.024,149.383
C00680=1146.998,-75.109,-44.856,178.982,6.024,149.382
C00681=1146.992,-74.859,-44.866,178.985,6.024,149.382
C00682=1146.987,-74.609,-44.876,178.987,6.025,149.381
C00683=1146.981,-74.360,-44.886,178.989,6.026,149.381
C00684=1146.977,-74.110,-44.896,178.991,6.026,149.380
C00685=1146.971,-73.860,-44.906,178.993,6.026,149.379
C00686=1146.966,-73.611,-44.917,178.996,6.027,149.379
C00687=1146.961,-73.361,-44.927,178.998,6.027,149.378
C00688=1146.955,-73.111,-44.937,179.000,6.027,149.378
C00689=1146.950,-72.862,-44.948,179.002,6.028,149.377
C00690=1146.945,-72.612,-44.958,179.005,6.029,149.377
C00691=1146.940,-72.362,-44.968,179.007,6.029,149.376
C00692=1146.934,-72.113,-44.978,179.009,6.029,149.376
C00693=1146.929,-71.863,-44.988,179.011,6.030,149.375
C00694=1146.924,-71.613,-44.999,179.013,6.031,149.374
C00695=1146.918,-71.363,-45.009,179.016,6.031,149.374
C00696=1146.912,-71.114,-45.019,179.017,6.031,149.374
C00697=1146.908,-70.864,-45.029,179.020,6.032,149.373
C00698=1146.902,-70.614,-45.039,179.022,6.032,149.372
C00699=1146.897,-70.365,-45.050,179.024,6.033,149.372
C00700=1146.892,-70.114,-45.060,179.026,6.033,149.371
C00701=1146.886,-69.865,-45.070,179.028,6.034,149.371
C00702=1146.881,-69.615,-45.081,179.031,6.034,149.370
C00703=1146.876,-69.365,-45.091,179.033,6.035,149.369
C00704=1146.870,-69.116,-45.101,179.036,6.035,149.369
C00705=1146.865,-68.865,-45.112,179.037,6.035,149.368
C00706=1146.859,-68.616,-45.122,179.040,6.036,149.368
C00707=1146.855,-68.367,-45.132,179.042,6.037,149.367
C00708=1146.850,-68.116,-45.142,179.044,6.037,149.367
C00709=1146.844,-67.867,-45.153,179.046,6.037,149.366
C00710=1146.839,-67.617,-45.164,179.048,6.038,149.366
C00711=1146.834,-67.368,-45.174,179.051,6.039,149.365
C00712=1146.828,-67.118,-45.184,179.053,6.039,149.364
C00713=1146.823,-66.868,-45.195,179.056,6.040,149.364
C00714=1146.818,-66.618,-45.205,179.057,6.040,149.363
C00715=1146.813,-66.368,-45.216,179.060,6.040,149.363
C00716=1146.807,-66.118,-45.226,179.062,6.041,149.362
C00717=1146.802,-65.870,-45.237,179.064,6.042,149.362
C00718=1146.797,-65.619,-45.247,179.067,6.042,149.361
C00719=1146.791,-65.370,-45.258,179.068,6.042,149.361
C00720=1146.786,-65.120,-45.268,179.071,6.043,149.360
C00721=1146.780,-64.870,-45.278,179.073,6.043,149.359
C00722=1146.775,-64.620,-45.289,179.075,6.044,149.359
C00723=1146.770,-64.371,-45.300,179.077,6.044,149.358
C00724=1146.765,-64.121,-45.310,179.080,6.044,149.358
C00725=1146.760,-63.871,-45.321,179.082,6.045,149.357
C00726=1146.754,-63.621,-45.331,179.084,6.046,149.357
C00727=1146.749,-63.372,-45.342,179.087,6.046,149.356
C00728=1146.744,-63.122,-45.352,179.088,6.046,149.356
C00729=1146.739,-62.872,-45.363,179.091,6.047,149.355
C00730=1146.733,-62.623,-45.373,179.093,6.047,149.354
C00731=1146.728,-62.373,-45.384,179.095,6.048,149.354
C00732=1146.723,-62.123,-45.395,179.098,6.049,149.353
C00733=1146.717,-61.874,-45.405,179.100,6.049,149.353
C00734=1146.712,-61.624,-45.415,179.102,6.049,149.352
C00735=1146.707,-61.375,-45.426,179.104,6.050,149.352
C00736=1146.702,-61.124,-45.437,179.107,6.050,149.351
C00737=1146.696,-60.875,-45.447,179.109,6.051,149.351
C00738=1146.691,-60.625,-45.459,179.112,6.052,149.350
C00739=1146.685,-60.375,-45.469,179.113,6.052,149.349
C00740=1146.680,-60.125,-45.480,179.115,6.052,149.349
C00741=1146.675,-59.876,-45.491,179.118,6.053,149.348
C00742=1146.670,-59.626,-45.501,179.120,6.054,149.348
C00743=1146.664,-59.376,-45.512,179.122,6.054,149.347
C00744=1146.660,-59.127,-45.523,179.125,6.055,149.347
C00745=1146.654,-58.877,-45.533,179.127,6.055,149.346
C00746=1146.649,-58.627,-45.544,179.129,6.055,149.346
C00747=1146.644,-58.378,-45.555,179.132,6.056,149.345
C00748=1146.638,-58.128,-45.566,179.134,6.057,149.344
C00749=1146.633,-57.878,-45.577,179.136,6.057,149.344
C00750=1146.628,-57.628,-45.587,179.138,6.057,149.343
C00751=1146.623,-57.378,-45.598,179.140,6.058,149.343
C00752=1146.618,-57.129,-45.609,179.142,6.059,149.342
C00753=1146.613,-56.879,-45.619,179.145,6.059,149.342
C00754=1146.607,-56.630,-45.630,179.147,6.060,149.341
C00755=1146.601,-56.379,-45.641,179.150,6.060,149.340
C00756=1146.596,-56.131,-45.652,179.152,6.061,149.340
C00757=1146.591,-55.880,-45.663,179.154,6.061,149.339
C00758=1146.587,-55.631,-45.674,179.156,6.061,149.339
C00759=1146.581,-55.381,-45.684,179.159,6.062,149.338
C00760=1146.575,-55.131,-45.696,179.161,6.063,149.338
C00761=1146.570,-54.882,-45.706,179.163,6.063,149.337
C00762=1146.565,-54.631,-45.717,179.166,6.064,149.337
C00763=1146.560,-54.382,-45.728,179.167,6.064,149.336
C00764=1146.555,-54.133,-45.739,179.170,6.064,149.335
C00765=1146.549,-53.882,-45.750,179.172,6.065,149.335
C00766=1146.544,-53.633,-45.761,179.175,6.066,149.334
C00767=1146.539,-53.383,-45.772,179.177,6.066,149.334
C00768=1146.534,-53.134,-45.783,179.179,6.067,149.333
C00769=1146.528,-52.884,-45.794,179.182,6.068,149.333
C00770=1146.523,-52.634,-45.805,179.183,6.068,149.332
C00771=1146.518,-52.384,-45.816,179.185,6.068,149.332
C00772=1146.513,-52.135,-45.827,179.188,6.069,149.331
C00773=1146.507,-51.885,-45.838,179.190,6.069,149.330
C00774=1146.502,-51.635,-45.849,179.193,6.070,149.330
C00775=1146.497,-51.386,-45.860,179.195,6.071,149.329
C00776=1146.492,-51.136,-45.870,179.197,6.071,149.329
C00777=1146.486,-50.865,-45.883,179.200,6.072,149.328
C00778=1146.480,-50.594,-45.895,179.202,6.073,149.328
C00779=1146.474,-50.324,-45.907,179.205,6.073,149.327
C00780=1146.468,-50.053,-45.919,179.208,6.073,149.326
C00781=1146.463,-49.804,-45.930,179.210,6.074,149.326
C00782=1146.458,-49.554,-45.941,179.212,6.075,149.325
C00783=1146.453,-49.304,-45.952,179.214,6.075,149.325
C00784=1146.447,-49.055,-45.963,179.216,6.075,149.324
C00785=1146.442,-48.805,-45.974,179.218,6.076,149.324
C00786=1146.437,-48.555,-45.986,179.221,6.077,149.323
C00787=1146.432,-48.306,-45.997,179.223,6.077,149.322
C00788=1146.427,-48.056,-46.007,179.226,6.078,149.322
C00789=1146.421,-47.806,-46.019,179.228,6.078,149.321
C00790=1146.416,-47.557,-46.030,179.230,6.079,149.321
C00791=1146.411,-47.307,-46.041,179.232,6.079,149.320
C00792=1146.406,-47.057,-46.053,179.235,6.080,149.320
C00793=1146.400,-46.808,-46.063,179.237,6.080,149.319
C00794=1146.395,-46.558,-46.075,179.239,6.081,149.318
C00795=1146.390,-46.307,-46.086,179.242,6.082,149.318
C00796=1146.385,-46.059,-46.097,179.244,6.082,149.317
C00797=1146.379,-45.809,-46.109,179.246,6.083,149.317
C00798=1146.374,-45.559,-46.120,179.249,6.084,149.316
C00799=1146.369,-45.309,-46.132,179.251,6.084,149.316
C00800=1146.363,-45.059,-46.142,179.254,6.085,149.315
C00801=1146.359,-44.810,-46.153,179.256,6.084,149.314
C00802=1146.353,-44.560,-46.165,179.258,6.085,149.314
C00803=1146.348,-44.311,-46.176,179.260,6.086,149.313
C00804=1146.342,-44.060,-46.187,179.263,6.086,149.313
C00805=1146.338,-43.811,-46.199,179.265,6.087,149.312
C00806=1146.332,-43.561,-46.211,179.267,6.088,149.312
C00807=1146.327,-43.312,-46.222,179.270,6.088,149.311
C00808=1146.321,-43.062,-46.233,179.272,6.089,149.311
C00809=1146.317,-42.812,-46.245,179.275,6.089,149.310
C00810=1146.312,-42.563,-46.256,179.277,6.090,149.309
C00811=1146.306,-42.313,-46.267,179.279,6.091,149.309
C00812=1146.301,-42.063,-46.278,179.281,6.091,149.308
C00813=1146.296,-41.813,-46.290,179.283,6.091,149.308
C00814=1146.291,-41.564,-46.301,179.286,6.092,149.307
C00815=1146.285,-41.314,-46.313,179.288,6.093,149.307
C00816=1146.280,-41.065,-46.324,179.290,6.093,149.306
C00817=1146.275,-40.815,-46.336,179.293,6.094,149.305
C00818=1146.270,-40.565,-46.347,179.295,6.095,149.305
C00819=1146.265,-40.315,-46.359,179.298,6.095,149.304
C00820=1146.259,-40.066,-46.371,179.300,6.096,149.304
C00821=1146.254,-39.816,-46.381,179.302,6.097,149.303
C00822=1146.248,-39.566,-46.393,179.305,6.097,149.303
C00823=1146.243,-39.316,-46.404,179.307,6.098,149.302
C00824=1146.238,-39.066,-46.416,179.310,6.098,149.301
C00825=1146.233,-38.817,-46.427,179.312,6.099,149.301
C00826=1146.227,-38.568,-46.439,179.313,6.099,149.300
C00827=1146.223,-38.318,-46.450,179.316,6.099,149.300
C00828=1146.217,-38.068,-46.462,179.318,6.100,149.299
C00829=1146.212,-37.818,-46.474,179.321,6.101,149.299
C00830=1146.206,-37.569,-46.485,179.323,6.101,149.298
C00831=1146.201,-37.319,-46.497,179.325,6.102,149.298
C00832=1146.196,-37.070,-46.508,179.328,6.103,149.297
C00833=1146.191,-36.820,-46.520,179.330,6.103,149.296
C00834=1146.186,-36.570,-46.532,179.333,6.104,149.296
C00835=1146.181,-36.320,-46.543,179.335,6.105,149.295
C00836=1146.175,-36.071,-46.556,179.337,6.105,149.295
C00837=1146.170,-35.821,-46.567,179.340,6.106,149.294
C00838=1146.165,-35.572,-46.579,179.342,6.107,149.294
C00839=1146.160,-35.322,-46.591,179.345,6.107,149.293
C00840=1146.155,-35.072,-46.602,179.347,6.108,149.292
C00841=1146.149,-34.822,-46.614,179.349,6.109,149.292
C00842=1146.144,-34.572,-46.626,179.352,6.109,149.291
C00843=1146.139,-34.324,-46.637,179.354,6.110,149.291
C00844=1146.133,-34.074,-46.648,179.357,6.110,149.290
C00845=1146.128,-33.824,-46.660,179.359,6.111,149.290
C00846=1146.123,-33.575,-46.672,179.361,6.111,149.289
C00847=1146.118,-33.325,-46.684,179.364,6.112,149.288
C00848=1146.113,-33.075,-46.696,179.366,6.113,149.288
C00849=1146.108,-32.825,-46.707,179.368,6.112,149.287
C00850=1146.102,-32.575,-46.719,179.370,6.113,149.287
C00851=1146.097,-32.325,-46.731,179.373,6.114,149.286
C00852=1146.091,-32.077,-46.743,179.375,6.114,149.286
C00853=1146.087,-31.827,-46.755,179.377,6.115,149.285
C00854=1146.081,-31.577,-46.767,179.380,6.116,149.284
C00855=1146.076,-31.327,-46.778,179.382,6.116,149.284
C00856=1146.071,-31.078,-46.790,179.385,6.117,149.283
C00857=1146.066,-30.828,-46.802,179.387,6.118,149.283
C00858=1146.061,-30.578,-46.814,179.389,6.118,149.282
C00859=1146.055,-30.328,-46.826,179.392,6.119,149.282
C00860=1146.050,-30.079,-46.837,179.394,6.120,149.281
C00861=1146.045,-29.829,-46.850,179.396,6.120,149.280
C00862=1146.040,-29.579,-46.862,179.399,6.121,149.280
C00863=1146.034,-29.329,-46.874,179.401,6.122,149.280
C00864=1146.030,-29.080,-46.885,179.403,6.122,149.279
C00865=1146.025,-28.831,-46.898,179.406,6.123,149.278
C00866=1146.019,-28.581,-46.910,179.408,6.123,149.278
C00867=1146.014,-28.331,-46.921,179.410,6.124,149.277
C00868=1146.009,-28.081,-46.934,179.413,6.124,149.276
C00869=1146.003,-27.832,-46.945,179.415,6.125,149.276
C00870=1145.998,-27.583,-46.957,179.417,6.126,149.276
C00871=1145.993,-27.333,-46.969,179.420,6.126,149.275
C00872=1145.987,-27.083,-46.981,179.422,6.127,149.274
C00873=1145.982,-26.833,-46.993,179.425,6.128,149.274
C00874=1145.978,-26.584,-47.005,179.427,6.128,149.273
C00875=1145.972,-26.334,-47.017,179.429,6.129,149.273
C00876=1145.967,-26.084,-47.029,179.432,6.130,149.272
C00877=1145.962,-25.835,-47.042,179.434,6.131,149.272
C00878=1145.956,-25.585,-47.053,179.437,6.131,149.271
C00879=1145.951,-25.336,-47.066,179.439,6.132,149.270
C00880=1145.946,-25.086,-47.078,179.442,6.132,149.270
C00881=1145.940,-24.816,-47.091,179.445,6.134,149.269
C00882=1145.935,-24.545,-47.104,179.447,6.134,149.269
C00883=1145.929,-24.276,-47.117,179.449,6.135,149.268
C00884=1145.924,-24.006,-47.130,179.452,6.135,149.267
C00885=1145.919,-23.756,-47.142,179.454,6.136,149.267
C00886=1145.913,-23.507,-47.155,179.457,6.137,149.266
C00887=1145.908,-23.257,-47.167,179.459,6.137,149.266
C00888=1145.903,-23.007,-47.179,179.462,6.138,149.265
C00889=1145.897,-22.757,-47.191,179.464,6.139,149.265
C00890=1145.892,-22.508,-47.204,179.467,6.139,149.264
C00891=1145.887,-22.258,-47.216,179.469,6.140,149.263
C00892=1145.882,-22.009,-47.228,179.471,6.141,149.263
C00893=1145.876,-21.759,-47.240,179.474,6.141,149.262
C00894=1145.871,-21.510,-47.253,179.476,6.142,149.262
C00895=1145.866,-21.259,-47.265,179.478,6.142,149.261
C00896=1145.861,-21.010,-47.277,179.481,6.144,149.261
C00897=1145.856,-20.760,-47.289,179.483,6.145,149.260
C00898=1145.851,-20.510,-47.302,179.486,6.145,149.259
C00899=1145.846,-20.261,-47.315,179.488,6.146,149.259
C00900=1145.840,-20.011,-47.326,179.491,6.146,149.258
C00901=1145.835,-19.762,-47.339,179.493,6.147,149.258
C00902=1145.830,-19.512,-47.351,179.496,6.147,149.257
C00903=1145.825,-19.263,-47.364,179.498,6.148,149.257
C00904=1145.819,-19.013,-47.375,179.500,6.149,149.256
C00905=1145.814,-18.763,-47.388,179.503,6.149,149.255
C00906=1145.809,-18.513,-47.401,179.505,6.150,149.255
C00907=1145.804,-18.263,-47.413,179.508,6.151,149.254
C00908=1145.799,-18.014,-47.425,179.510,6.151,149.254
C00909=1145.794,-17.765,-47.438,179.512,6.152,149.253
C00910=1145.788,-17.515,-47.450,179.515,6.153,149.253
C00911=1145.783,-17.265,-47.463,179.517,6.153,149.252
C00912=1145.778,-17.016,-47.475,179.519,6.154,149.251
C00913=1145.773,-16.765,-47.487,179.522,6.155,149.251
C00914=1145.768,-16.516,-47.500,179.525,6.156,149.250
C00915=1145.763,-16.267,-47.513,179.527,6.157,149.250
C00916=1145.758,-16.017,-47.524,179.529,6.158,149.249
C00917=1145.752,-15.768,-47.537,179.532,6.158,149.249
C00918=1145.747,-15.518,-47.550,179.534,6.159,149.248
C00919=1145.742,-15.269,-47.562,179.537,6.159,149.248
C00920=1145.737,-15.018,-47.575,179.539,6.160,149.247
C00921=1145.732,-14.769,-47.588,179.542,6.160,149.246
C00922=1145.726,-14.519,-47.600,179.544,6.161,149.246
C00923=1145.721,-14.270,-47.613,179.546,6.162,149.245
C00924=1145.716,-14.020,-47.625,179.549,6.162,149.245
C00925=1145.711,-13.770,-47.638,179.551,6.163,149.244
C00926=1145.706,-13.521,-47.650,179.553,6.164,149.244
C00927=1145.701,-13.271,-47.663,179.556,6.165,149.243
C00928=1145.696,-13.022,-47.676,179.559,6.166,149.242
C00929=1145.690,-12.772,-47.688,179.561,6.166,149.242
C00930=1145.685,-12.522,-47.701,179.563,6.167,149.241
C00931=1145.680,-12.273,-47.714,179.566,6.168,149.241
C00932=1145.675,-12.023,-47.726,179.568,6.168,149.240
C00933=1145.670,-11.774,-47.739,179.571,6.169,149.240
C00934=1145.665,-11.524,-47.752,179.573,6.170,149.239
C00935=1145.659,-11.274,-47.764,179.576,6.170,149.238
C00936=1145.654,-11.024,-47.777,179.578,6.171,149.238
C00937=1145.649,-10.775,-47.789,179.581,6.173,149.238
C00938=1145.644,-10.526,-47.802,179.583,6.173,149.237
C00939=1145.639,-10.276,-47.815,179.585,6.174,149.236
C00940=1145.633,-10.026,-47.828,179.588,6.174,149.236
C00941=1145.628,-9.777,-47.841,179.590,6.175,149.235
C00942=1145.624,-9.527,-47.854,179.593,6.175,149.235
C00943=1145.619,-9.277,-47.866,179.595,6.176,149.234
C00944=1145.613,-9.028,-47.880,179.597,6.177,149.234
C00945=1145.607,-8.778,-47.892,179.600,6.177,149.233
C00946=1145.603,-8.528,-47.904,179.603,6.179,149.232
C00947=1145.598,-8.279,-47.917,179.605,6.179,149.232
C00948=1145.592,-8.029,-47.930,179.607,6.180,149.231
C00949=1145.587,-7.780,-47.943,179.610,6.181,149.231
C00950=1145.582,-7.530,-47.956,179.612,6.182,149.230
C00951=1145.577,-7.280,-47.968,179.615,6.182,149.230
C00952=1145.571,-7.031,-47.982,179.617,6.183,149.229
C00953=1145.567,-6.781,-47.995,179.619,6.184,149.228
C00954=1145.562,-6.531,-48.007,179.623,6.185,149.228
C00955=1145.556,-6.282,-48.020,179.625,6.186,149.227
C00956=1145.551,-6.032,-48.033,179.627,6.186,149.227
C00957=1145.546,-5.783,-48.047,179.630,6.187,149.226
C00958=1145.541,-5.533,-48.060,179.632,6.188,149.226
C00959=1145.536,-5.283,-48.073,179.634,6.188,149.225
C00960=1145.531,-5.034,-48.085,179.637,6.189,149.225
C00961=1145.525,-4.784,-48.099,179.640,6.190,149.224
C00962=1145.521,-4.534,-48.112,179.642,6.191,149.223
C00963=1145.515,-4.285,-48.124,179.645,6.191,149.223
C00964=1145.510,-4.035,-48.137,179.647,6.192,149.222
C00965=1145.505,-3.785,-48.150,179.649,6.193,149.222
C00966=1145.500,-3.536,-48.163,179.652,6.193,149.221
C00967=1145.494,-3.286,-48.176,179.654,6.194,149.221
C00968=1145.490,-3.037,-48.190,179.657,6.195,149.220
C00969=1145.484,-2.787,-48.203,179.659,6.196,149.219
C00970=1145.479,-2.538,-48.216,179.662,6.197,149.219
C00971=1145.474,-2.288,-48.229,179.664,6.197,149.218
C00972=1145.468,-2.038,-48.242,179.666,6.198,149.218
C00973=1145.464,-1.788,-48.255,179.669,6.199,149.217
C00974=1145.458,-1.539,-48.269,179.672,6.200,149.217
C00975=1145.453,-1.290,-48.281,179.674,6.201,149.216
C00976=1145.449,-1.040,-48.294,179.677,6.202,149.216
C00977=1145.443,-0.790,-48.307,179.679,6.202,149.215
C00978=1145.438,-0.540,-48.320,179.681,6.203,149.214
C00979=1145.433,-0.291,-48.334,179.684,6.204,149.214
C00980=1145.428,-0.042,-48.347,179.687,6.205,149.213
C00981=1145.422,0.208,-48.360,179.689,6.206,149.213
C00982=1145.417,0.458,-48.373,179.692,6.206,149.212
C00983=1145.412,0.707,-48.387,179.694,6.207,149.212
C00984=1145.407,0.957,-48.400,179.697,6.207,149.211
C00985=1145.401,1.227,-48.414,179.699,6.209,149.210
C00986=1145.395,1.495,-48.429,179.702,6.209,149.210
C00987=1145.390,1.765,-48.443,179.704,6.210,149.209
C00988=1145.385,2.035,-48.458,179.707,6.211,149.209
C00989=1145.380,2.284,-48.470,179.710,6.212,149.208
C00990=1145.375,2.534,-48.484,179.712,6.213,149.207
C00991=1145.370,2.783,-48.497,179.714,6.213,149.207
C00992=1145.365,3.033,-48.511,179.717,6.214,149.206
C00993=1145.359,3.282,-48.524,179.720,6.216,149.206
C00994=1145.354,3.532,-48.537,179.722,6.216,149.205
C00995=1145.349,3.782,-48.551,179.725,6.217,149.205
C00996=1145.344,4.031,-48.564,179.727,6.217,149.204
C00997=1145.338,4.281,-48.578,179.729,6.218,149.204
C00998=1145.334,4.530,-48.591,179.732,6.220,149.203
C00999=1145.328,4.780,-48.604,179.735,6.220,149.202
C01000=1145.324,5.030,-48.617,179.737,6.221,149.202
C01001=1145.318,5.279,-48.631,179.740,6.221,149.201
C01002=1145.313,5.529,-48.645,179.742,6.222,149.201
C01003=1145.308,5.778,-48.658,179.745,6.224,149.200
C01004=1145.303,6.028,-48.672,179.747,6.224,149.200
C01005=1145.298,6.277,-48.685,179.750,6.225,149.199
C01006=1145.293,6.527,-48.699,179.752,6.225,149.198
C01007=1145.287,6.776,-48.713,179.755,6.227,149.198
C01008=1145.283,7.026,-48.725,179.758,6.227,149.197
C01009=1145.277,7.275,-48.739,179.760,6.228,149.197
C01010=1145.272,7.526,-48.753,179.762,6.229,149.196
C01011=1145.267,7.774,-48.766,179.765,6.230,149.196
C01012=1145.262,8.025,-48.780,179.767,6.231,149.195
C01013=1145.256,8.274,-48.794,179.770,6.232,149.195
C01014=1145.252,8.524,-48.807,179.772,6.232,149.194
C01015=1145.246,8.773,-48.821,179.775,6.233,149.193
C01016=1145.241,9.023,-48.834,179.778,6.234,149.193
C01017=1145.237,9.272,-48.848,179.780,6.235,149.192
C01018=1145.231,9.522,-48.861,179.782,6.236,149.192
C01019=1145.226,9.772,-48.875,179.785,6.237,149.191
C01020=1145.221,10.021,-48.889,179.787,6.237,149.191
C01021=1145.216,10.271,-48.902,179.790,6.239,149.190
C01022=1145.210,10.520,-48.916,179.793,6.239,149.190
C01023=1145.205,10.770,-48.930,179.795,6.240,149.189
C01024=1145.201,11.020,-48.943,179.797,6.241,149.189
C01025=1145.195,11.269,-48.957,179.800,6.242,149.188
C01026=1145.190,11.519,-48.971,179.802,6.243,149.187
C01027=1145.185,11.768,-48.984,179.805,6.243,149.187
C01028=1145.180,12.017,-48.998,179.807,6.244,149.186
C01029=1145.175,12.268,-49.012,179.811,6.245,149.186
C01030=1145.169,12.517,-49.026,179.813,6.246,149.185
C01031=1145.165,12.766,-49.040,179.815,6.247,149.185
C01032=1145.160,13.016,-49.053,179.818,6.247,149.184
C01033=1145.154,13.265,-49.067,179.820,6.249,149.184
C01034=1145.150,13.515,-49.081,179.823,6.249,149.183
C01035=1145.144,13.765,-49.095,179.825,6.250,149.182
C01036=1145.139,14.014,-49.108,179.827,6.251,149.182
C01037=1145.134,14.264,-49.123,179.831,6.252,149.181
C01038=1145.129,14.513,-49.136,179.833,6.253,149.181
C01039=1145.124,14.763,-49.150,179.835,6.253,149.180
C01040=1145.119,15.013,-49.164,179.838,6.255,149.180
C01041=1145.113,15.262,-49.178,179.841,6.256,149.179
C01042=1145.109,15.511,-49.192,179.843,6.256,149.179
C01043=1145.104,15.761,-49.206,179.845,6.257,149.178
C01044=1145.098,16.011,-49.219,179.848,6.258,149.177
C01045=1145.093,16.260,-49.234,179.851,6.259,149.177
C01046=1145.088,16.510,-49.248,179.853,6.260,149.176
C01047=1145.083,16.759,-49.262,179.855,6.261,149.176
C01048=1145.078,17.009,-49.276,179.859,6.262,149.175
C01049=1145.073,17.258,-49.290,179.861,6.263,149.175
C01050=1145.068,17.509,-49.303,179.863,6.263,149.174
C01051=1145.063,17.758,-49.317,179.866,6.265,149.173
C01052=1145.058,18.007,-49.331,179.868,6.265,149.173
C01053=1145.053,18.257,-49.346,179.871,6.266,149.172
C01054=1145.047,18.506,-49.360,179.874,6.268,149.172
C01055=1145.042,18.756,-49.374,179.876,6.268,149.171
C01056=1145.037,19.005,-49.388,179.879,6.269,149.171
C01057=1145.032,19.255,-49.403,179.881,6.270,149.170
C01058=1145.027,19.504,-49.416,179.884,6.271,149.170
C01059=1145.022,19.754,-49.431,179.886,6.272,149.169
C01060=1145.017,20.004,-49.445,179.889,6.272,149.168
C01061=1145.012,20.254,-49.459,179.892,6.274,149.168
C01062=1145.006,20.503,-49.472,179.894,6.275,149.168
C01063=1145.001,20.753,-49.487,179.896,6.275,149.167
C01064=1144.996,21.002,-49.501,179.899,6.277,149.166
C01065=1144.991,21.252,-49.515,179.902,6.277,149.166
C01066=1144.986,21.501,-49.529,179.904,6.278,149.165
C01067=1144.981,21.751,-49.543,179.906,6.279,149.165
C01068=1144.976,22.000,-49.558,179.909,6.280,149.164
C01069=1144.971,22.250,-49.572,179.912,6.281,149.164
C01070=1144.965,22.499,-49.586,179.914,6.281,149.163
C01071=1144.961,22.748,-49.601,179.917,6.283,149.163
C01072=1144.956,22.998,-49.615,179.920,6.283,149.162
C01073=1144.951,23.248,-49.629,179.922,6.284,149.161
C01074=1144.946,23.497,-49.644,179.925,6.286,149.161
C01075=1144.940,23.746,-49.658,179.927,6.286,149.160
C01076=1144.935,23.996,-49.672,179.929,6.287,149.160
C01077=1144.930,24.246,-49.686,179.933,6.288,149.159
C01078=1144.925,24.496,-49.701,179.935,6.289,149.159
C01079=1144.920,24.745,-49.715,179.937,6.290,149.158
C01080=1144.915,24.995,-49.729,179.940,6.291,149.158
C01081=1144.910,25.243,-49.744,179.942,6.292,149.157
C01082=1144.905,25.493,-49.758,179.945,6.293,149.156
C01083=1144.900,25.743,-49.772,179.948,6.294,149.156
C01084=1144.895,25.992,-49.787,179.950,6.295,149.156
C01085=1144.890,26.242,-49.801,179.953,6.295,149.155
C01086=1144.885,26.492,-49.816,179.955,6.297,149.154
C01087=1144.880,26.741,-49.831,179.958,6.297,149.154
C01088=1144.874,26.990,-49.845,179.960,6.298,149.153
C01089=1144.869,27.260,-49.860,179.963,6.300,149.153
C01090=1144.864,27.528,-49.875,179.966,6.301,149.152
C01091=1144.858,27.798,-49.892,179.969,6.302,149.151
C01092=1144.853,28.066,-49.907,179.972,6.303,149.151
C01093=1144.848,28.316,-49.922,179.974,6.304,149.150
C01094=1144.843,28.566,-49.936,179.976,6.305,149.150
C01095=1144.838,28.816,-49.950,179.980,6.306,149.149
C01096=1144.832,29.064,-49.965,179.982,6.307,149.149
C01097=1144.827,29.314,-49.980,179.984,6.307,149.148
C01098=1144.822,29.564,-49.994,179.987,6.309,149.148
C01099=1144.817,29.813,-50.009,179.989,6.310,149.147
C01100=1144.812,30.062,-50.023,179.993,6.311,149.146
C01101=1144.807,30.312,-50.038,179.995,6.312,149.146
C01102=1144.802,30.562,-50.053,179.997,6.312,149.146
C01103=1144.797,30.811,-50.067,-180.000,6.314,149.145
C01104=1144.792,31.061,-50.082,-179.998,6.315,149.144
C01105=1144.787,31.310,-50.097,-179.995,6.315,149.144
C01106=1144.782,31.560,-50.111,-179.992,6.317,149.143
C01107=1144.777,31.810,-50.126,-179.990,6.317,149.143
C01108=1144.772,32.059,-50.141,-179.987,6.319,149.142
C01109=1144.767,32.309,-50.156,-179.985,6.320,149.142
C01110=1144.762,32.558,-50.171,-179.982,6.320,149.141
C01111=1144.756,32.807,-50.184,-179.979,6.322,149.141
C01112=1144.751,33.057,-50.199,-179.977,6.322,149.140
C01113=1144.746,33.306,-50.214,-179.974,6.323,149.139
C01114=1144.741,33.556,-50.229,-179.972,6.325,149.139
C01115=1144.736,33.805,-50.244,-179.969,6.325,149.138
C01116=1144.731,34.055,-50.258,-179.966,6.327,149.138
C01117=1144.726,34.304,-50.273,-179.964,6.327,149.137
C01118=1144.721,34.554,-50.288,-179.961,6.328,149.137
C01119=1144.716,34.803,-50.303,-179.959,6.330,149.136
C01120=1144.711,35.053,-50.318,-179.956,6.330,149.136
C01121=1144.706,35.302,-50.333,-179.953,6.332,149.135
C01122=1144.700,35.552,-50.347,-179.951,6.333,149.135
C01123=1144.696,35.801,-50.362,-179.948,6.333,149.134
C01124=1144.691,36.051,-50.377,-179.946,6.335,149.134
C01125=1144.685,36.300,-50.392,-179.943,6.335,149.133
C01126=1144.681,36.550,-50.407,-179.940,6.337,149.132
C01127=1144.675,36.799,-50.422,-179.938,6.338,149.132
C01128=1144.670,37.049,-50.436,-179.935,6.339,149.131
C01129=1144.666,37.299,-50.452,-179.933,6.340,149.131
C01130=1144.661,37.548,-50.467,-179.930,6.340,149.130
C01131=1144.656,37.798,-50.482,-179.927,6.342,149.130
C01132=1144.650,38.047,-50.497,-179.925,6.343,149.129
C01133=1144.645,38.297,-50.512,-179.922,6.344,149.129
C01134=1144.640,38.546,-50.527,-179.920,6.345,149.128
C01135=1144.635,38.796,-50.542,-179.917,6.346,149.128
C01136=1144.630,39.045,-50.556,-179.914,6.347,149.127
C01137=1144.625,39.295,-50.572,-179.912,6.348,149.127
C01138=1144.620,39.544,-50.587,-179.909,6.349,149.126
C01139=1144.615,39.794,-50.602,-179.907,6.350,149.126
C01140=1144.610,40.043,-50.617,-179.904,6.351,149.125
C01141=1144.605,40.292,-50.632,-179.901,6.352,149.124
C01142=1144.600,40.542,-50.647,-179.899,6.353,149.124
C01143=1144.594,40.791,-50.662,-179.896,6.354,149.123
C01144=1144.590,41.041,-50.678,-179.894,6.355,149.123
C01145=1144.585,41.291,-50.693,-179.891,6.356,149.122
C01146=1144.580,41.540,-50.708,-179.888,6.357,149.122
C01147=1144.575,41.790,-50.723,-179.886,6.358,149.121
C01148=1144.570,42.039,-50.738,-179.883,6.359,149.121
C01149=1144.565,42.288,-50.754,-179.880,6.361,149.120
C01150=1144.560,42.538,-50.768,-179.878,6.361,149.120
C01151=1144.554,42.787,-50.784,-179.875,6.363,149.119
C01152=1144.549,43.037,-50.800,-179.873,6.363,149.119
C01153=1144.545,43.286,-50.815,-179.870,6.365,149.118
C01154=1144.539,43.536,-50.830,-179.867,6.366,149.117
C01155=1144.534,43.786,-50.844,-179.865,6.366,149.117
C01156=1144.529,44.035,-50.860,-179.862,6.368,149.117
C01157=1144.524,44.284,-50.875,-179.860,6.369,149.116
C01158=1144.520,44.534,-50.891,-179.857,6.370,149.115
C01159=1144.514,44.784,-50.907,-179.854,6.371,149.115
C01160=1144.510,45.033,-50.922,-179.852,6.372,149.114
C01161=1144.504,45.282,-50.937,-179.849,6.373,149.114
C01162=1144.500,45.531,-50.952,-179.846,6.374,149.113
C01163=1144.494,45.781,-50.967,-179.844,6.375,149.113
C01164=1144.489,46.031,-50.983,-179.841,6.377,149.112
C01165=1144.484,46.280,-50.998,-179.839,6.377,149.112
C01166=1144.479,46.530,-51.014,-179.836,6.379,149.111
C01167=1144.474,46.779,-51.029,-179.833,6.379,149.111
C01168=1144.469,47.028,-51.044,-179.830,6.381,149.110
C01169=1144.464,47.278,-51.060,-179.828,6.382,149.110
C01170=1144.459,47.528,-51.076,-179.825,6.383,149.109
C01171=1144.454,47.777,-51.091,-179.823,6.384,149.109
C01172=1144.449,48.026,-51.106,-179.820,6.386,149.108
C01173=1144.444,48.276,-51.122,-179.818,6.386,149.107
C01174=1144.439,48.525,-51.137,-179.815,6.388,149.107
C01175=1144.434,48.775,-51.153,-179.813,6.389,149.107
C01176=1144.429,49.024,-51.168,-179.809,6.390,149.106
C01177=1144.425,49.274,-51.184,-179.807,6.391,149.105
C01178=1144.419,49.523,-51.199,-179.804,6.392,149.105
C01179=1144.414,49.773,-51.215,-179.802,6.393,149.104
C01180=1144.408,50.022,-51.230,-179.799,6.395,149.104
C01181=1144.404,50.272,-51.246,-179.796,6.395,149.103
C01182=1144.399,50.521,-51.261,-179.794,6.397,149.103
C01183=1144.394,50.770,-51.278,-179.791,6.397,149.102
C01184=1144.390,51.020,-51.293,-179.788,6.399,149.102
C01185=1144.384,51.269,-51.309,-179.786,6.400,149.101
C01186=1144.379,51.519,-51.324,-179.783,6.401,149.101
C01187=1144.374,51.768,-51.340,-179.781,6.402,149.100
C01188=1144.369,52.018,-51.356,-179.778,6.403,149.100
C01189=1144.364,52.267,-51.371,-179.776,6.404,149.099
C01190=1144.359,52.516,-51.387,-179.773,6.405,149.099
C01191=1144.354,52.766,-51.403,-179.770,6.406,149.098
C01192=1144.349,53.016,-51.419,-179.768,6.408,149.098
C01193=1144.343,53.284,-51.436,-179.764,6.409,149.097
C01194=1144.338,53.553,-51.453,-179.762,6.410,149.096
C01195=1144.332,53.821,-51.470,-179.759,6.411,149.096
C01196=1144.328,54.090,-51.486,-179.756,6.413,149.095
C01197=1144.323,54.339,-51.502,-179.754,6.413,149.095
C01198=1144.317,54.589,-51.518,-179.751,6.415,149.094
C01199=1144.312,54.839,-51.534,-179.748,6.416,149.094
C01200=1144.307,55.088,-51.550,-179.745,6.417,149.093
C01201=1144.302,55.337,-51.565,-179.743,6.418,149.093
C01202=1144.297,55.587,-51.581,-179.740,6.419,149.092
C01203=1144.292,55.837,-51.597,-179.737,6.421,149.092
C01204=1144.287,56.085,-51.613,-179.735,6.422,149.091
C01205=1144.283,56.335,-51.629,-179.732,6.423,149.091
C01206=1144.277,56.585,-51.644,-179.730,6.424,149.090
C01207=1144.273,56.834,-51.661,-179.727,6.426,149.090
C01208=1144.267,57.084,-51.677,-179.724,6.426,149.089
C01209=1144.262,57.333,-51.692,-179.722,6.428,149.089
C01210=1144.258,57.582,-51.709,-179.719,6.429,149.088
C01211=1144.252,57.832,-51.724,-179.716,6.430,149.087
C01212=1144.248,58.081,-51.741,-179.714,6.432,149.087
C01213=1144.242,58.331,-51.757,-179.711,6.432,149.087
C01214=1144.237,58.580,-51.772,-179.708,6.434,149.086
C01215=1144.232,58.830,-51.789,-179.706,6.434,149.085
C01216=1144.227,59.079,-51.804,-179.703,6.436,149.085
C01217=1144.223,59.328,-51.821,-179.701,6.437,149.084
C01218=1144.217,59.578,-51.837,-179.698,6.438,149.084
C01219=1144.212,59.828,-51.853,-179.695,6.440,149.084
C01220=1144.207,60.077,-51.869,-179.692,6.440,149.083
C01221=1144.202,60.326,-51.885,-179.690,6.442,149.082
C01222=1144.197,60.576,-51.901,-179.688,6.443,149.082
C01223=1144.192,60.825,-51.917,-179.684,6.444,149.081
C01224=1144.188,61.075,-51.934,-179.682,6.446,149.081
C01225=1144.182,61.324,-51.949,-179.679,6.447,149.080
C01226=1144.178,61.573,-51.966,-179.676,6.448,149.080
C01227=1144.172,61.823,-51.981,-179.674,6.449,149.079
C01228=1144.168,62.072,-51.998,-179.671,6.450,149.079
C01229=1144.163,62.321,-52.014,-179.669,6.451,149.078
C01230=1144.158,62.571,-52.030,-179.666,6.453,149.078
C01231=1144.153,62.820,-52.047,-179.663,6.454,149.077
C01232=1144.148,63.070,-52.063,-179.661,6.455,149.077
C01233=1144.142,63.319,-52.079,-179.658,6.456,149.076
C01234=1144.138,63.569,-52.095,-179.656,6.457,149.076
C01235=1144.132,63.818,-52.112,-179.652,6.459,149.075
C01236=1144.128,64.068,-52.128,-179.650,6.460,149.075
C01237=1144.123,64.317,-52.144,-179.647,6.461,149.074
C01238=1144.118,64.566,-52.161,-179.644,6.462,149.074
C01239=1144.113,64.815,-52.177,-179.641,6.464,149.073
C01240=1144.108,65.065,-52.193,-179.639,6.465,149.073
C01241=1144.102,65.314,-52.210,-179.636,6.466,149.072
C01242=1144.098,65.564,-52.226,-179.634,6.467,149.072
C01243=1144.093,65.814,-52.242,-179.631,6.469,149.071
C01244=1144.088,66.063,-52.259,-179.628,6.470,149.071
C01245=1144.084,66.312,-52.275,-179.626,6.471,149.070
C01246=1144.078,66.562,-52.291,-179.623,6.472,149.070
C01247=1144.073,66.811,-52.308,-179.620,6.474,149.069
C01248=1144.068,67.060,-52.325,-179.618,6.475,149.069
C01249=1144.063,67.310,-52.341,-179.615,6.476,149.068
C01250=1144.059,67.560,-52.357,-179.613,6.477,149.068
C01251=1144.054,67.809,-52.373,-179.610,6.478,149.067
C01252=1144.048,68.058,-52.391,-179.607,6.480,149.067
C01253=1144.043,68.307,-52.407,-179.605,6.481,149.066
C01254=1144.039,68.557,-52.424,-179.601,6.482,149.066
C01255=1144.034,68.807,-52.440,-179.599,6.484,149.065
C01256=1144.028,69.056,-52.457,-179.597,6.485,149.065
C01257=1144.024,69.305,-52.473,-179.594,6.486,149.064
C01258=1144.019,69.554,-52.490,-179.591,6.488,149.064
C01259=1144.014,69.804,-52.506,-179.588,6.488,149.063
C01260=1144.009,70.053,-52.523,-179.586,6.490,149.063
C01261=1144.004,70.303,-52.539,-179.583,6.491,149.062
C01262=1143.999,70.552,-52.556,-179.580,6.492,149.062
C01263=1143.994,70.802,-52.573,-179.578,6.494,149.061
C01264=1143.989,71.051,-52.589,-179.575,6.494,149.061
C01265=1143.984,71.300,-52.606,-179.572,6.496,149.060
C01266=1143.979,71.550,-52.623,-179.569,6.498,149.060
C01267=1143.974,71.799,-52.640,-179.567,6.499,149.059
C01268=1143.969,72.048,-52.656,-179.564,6.500,149.059
C01269=1143.964,72.298,-52.673,-179.561,6.502,149.058
C01270=1143.959,72.547,-52.690,-179.559,6.502,149.058
C01271=1143.955,72.796,-52.706,-179.556,6.504,149.057
C01272=1143.950,73.046,-52.724,-179.553,6.505,149.057
C01273=1143.944,73.295,-52.740,-179.551,6.506,149.056
C01274=1143.940,73.545,-52.757,-179.548,6.508,149.056
C01275=1143.935,73.794,-52.774,-179.545,6.509,149.055
C01276=1143.930,74.043,-52.790,-179.543,6.510,149.055
C01277=1143.924,74.293,-52.807,-179.540,6.512,149.054
C01278=1143.920,74.542,-52.824,-179.537,6.513,149.054
C01279=1143.915,74.791,-52.840,-179.534,6.515,149.053
C01280=1143.910,75.041,-52.858,-179.532,6.515,149.053
C01281=1143.905,75.290,-52.874,-179.529,6.517,149.052
C01282=1143.900,75.540,-52.892,-179.526,6.518,149.052
C01283=1143.895,75.789,-52.908,-179.524,6.519,149.051
C01284=1143.890,76.039,-52.925,-179.521,6.521,149.051
C01285=1143.885,76.288,-52.942,-179.518,6.522,149.050
C01286=1143.880,76.538,-52.959,-179.516,6.523,149.050
C01287=1143.875,76.786,-52.976,-179.513,6.525,149.049
C01288=1143.870,77.036,-52.993,-179.510,6.526,149.049
C01289=1143.865,77.286,-53.010,-179.508,6.527,149.048
C01290=1143.860,77.535,-53.027,-179.505,6.529,149.048
C01291=1143.855,77.784,-53.044,-179.502,6.530,149.047
C01292=1143.850,78.034,-53.061,-179.499,6.532,149.047
C01293=1143.846,78.283,-53.078,-179.497,6.532,149.046
C01294=1143.841,78.533,-53.096,-179.494,6.534,149.046
C01295=1143.836,78.782,-53.112,-179.491,6.536,149.045
C01296=1143.830,79.031,-53.129,-179.489,6.537,149.045
C01297=1143.826,79.300,-53.147,-179.486,6.538,149.044
C01298=1143.820,79.569,-53.166,-179.483,6.540,149.044
C01299=1143.815,79.836,-53.185,-179.480,6.541,149.043
C01300=1143.810,80.105,-53.203,-179.477,6.543,149.043
C01301=1143.805,80.355,-53.220,-179.475,6.544,149.042
C01302=1143.800,80.603,-53.237,-179.471,6.545,149.042
C01303=1143.795,80.852,-53.255,-179.469,6.546,149.041
C01304=1143.789,81.102,-53.272,-179.466,6.548,149.041
C01305=1143.785,81.352,-53.289,-179.464,6.550,149.040
C01306=1143.780,81.602,-53.306,-179.460,6.551,149.040
C01307=1143.776,81.850,-53.323,-179.458,6.552,149.039
C01308=1143.770,82.099,-53.340,-179.456,6.554,149.039
C01309=1143.765,82.349,-53.358,-179.452,6.555,149.038
C01310=1143.760,82.598,-53.375,-179.450,6.556,149.038
C01311=1143.755,82.848,-53.392,-179.447,6.557,149.037
C01312=1143.750,83.097,-53.410,-179.445,6.559,149.037
C01313=1143.746,83.347,-53.427,-179.442,6.561,149.037
C01314=1143.741,83.596,-53.444,-179.439,6.562,149.036
C01315=1143.736,83.846,-53.462,-179.437,6.563,149.035
C01316=1143.731,84.094,-53.478,-179.434,6.565,149.035
C01317=1143.726,84.344,-53.496,-179.431,6.566,149.035
C01318=1143.720,84.593,-53.513,-179.428,6.567,149.034
C01319=1143.716,84.842,-53.531,-179.426,6.568,149.034
C01320=1143.711,85.092,-53.548,-179.423,6.570,149.033
C01321=1143.706,85.341,-53.566,-179.420,6.572,149.033
C01322=1143.702,85.591,-53.583,-179.417,6.573,149.032
C01323=1143.697,85.840,-53.601,-179.415,6.574,149.032
C01324=1143.692,86.090,-53.618,-179.412,6.576,149.031
C01325=1143.687,86.339,-53.636,-179.409,6.577,149.031
C01326=1143.682,86.588,-53.653,-179.406,6.578,149.030
C01327=1143.677,86.837,-53.670,-179.404,6.579,149.030
C01328=1143.671,87.087,-53.688,-179.401,6.581,149.029
C01329=1143.666,87.336,-53.706,-179.399,6.583,149.029
C01330=1143.662,87.585,-53.723,-179.395,6.584,149.028
C01331=1143.657,87.834,-53.740,-179.393,6.586,149.028
C01332=1143.652,88.084,-53.758,-179.390,6.587,149.027
C01333=1143.647,88.333,-53.775,-179.388,6.588,149.027
C01334=1143.642,88.583,-53.793,-179.385,6.590,149.027
C01335=1143.637,88.832,-53.811,-179.382,6.591,149.026
C01336=1143.633,89.081,-53.828,-179.380,6.592,149.025
C01337=1143.628,89.330,-53.846,-179.377,6.594,149.025
C01338=1143.623,89.580,-53.864,-179.374,6.595,149.025
C01339=1143.618,89.829,-53.881,-179.371,6.597,149.024
C01340=1143.613,90.079,-53.899,-179.368,6.598,149.024
C01341=1143.608,90.328,-53.917,-179.366,6.599,149.023
C01342=1143.603,90.577,-53.934,-179.363,6.601,149.023
C01343=1143.598,90.826,-53.952,-179.361,6.603,149.022
C01344=1143.593,91.076,-53.970,-179.357,6.604,149.022
C01345=1143.588,91.325,-53.987,-179.355,6.606,149.021
C01346=1143.583,91.574,-54.005,-179.353,6.606,149.021
C01347=1143.578,91.824,-54.023,-179.350,6.608,149.020
C01348=1143.574,92.073,-54.041,-179.347,6.610,149.020
C01349=1143.569,92.322,-54.059,-179.344,6.611,149.019
C01350=1143.563,92.572,-54.076,-179.341,6.613,149.019
C01351=1143.558,92.821,-54.094,-179.338,6.614,149.018
C01352=1143.554,93.071,-54.113,-179.336,6.615,149.018
C01353=1143.550,93.320,-54.130,-179.333,6.617,149.018
C01354=1143.545,93.569,-54.148,-179.330,6.618,149.017
C01355=1143.540,93.819,-54.165,-179.328,6.620,149.017
C01356=1143.535,94.068,-54.183,-179.325,6.622,149.016
C01357=1143.530,94.317,-54.201,-179.323,6.623,149.016
C01358=1143.525,94.566,-54.219,-179.320,6.624,149.015
C01359=1143.520,94.815,-54.237,-179.317,6.625,149.015
C01360=1143.515,95.065,-54.255,-179.314,6.627,149.014
C01361=1143.510,95.314,-54.273,-179.311,6.629,149.014
C01362=1143.505,95.563,-54.291,-179.308,6.631,149.013
C01363=1143.500,95.813,-54.308,-179.306,6.632,149.013
C01364=1143.496,96.063,-54.327,-179.303,6.633,149.012
C01365=1143.491,96.312,-54.345,-179.300,6.634,149.012
C01366=1143.486,96.561,-54.363,-179.298,6.636,149.012
C01367=1143.480,96.810,-54.381,-179.295,6.638,149.011
C01368=1143.476,97.060,-54.399,-179.292,6.639,149.011
C01369=1143.471,97.309,-54.417,-179.289,6.641,149.010
C01370=1143.466,97.558,-54.435,-179.287,6.642,149.010
C01371=1143.461,97.807,-54.453,-179.284,6.643,149.009
C01372=1143.457,98.057,-54.472,-179.281,6.645,149.009
C01373=1143.452,98.306,-54.489,-179.279,6.647,149.008
C01374=1143.447,98.555,-54.507,-179.276,6.648,149.008
C01375=1143.442,98.805,-54.525,-179.273,6.650,149.007
C01376=1143.437,99.054,-54.543,-179.270,6.651,149.007
C01377=1143.432,99.302,-54.562,-179.268,6.652,149.006
C01378=1143.427,99.552,-54.581,-179.265,6.654,149.006
C01379=1143.422,99.802,-54.599,-179.262,6.656,149.006
C01380=1143.417,100.051,-54.617,-179.260,6.657,149.005
C01381=1143.412,100.300,-54.635,-179.256,6.659,149.005
C01382=1143.408,100.549,-54.653,-179.254,6.660,149.004
C01383=1143.403,100.799,-54.671,-179.251,6.662,149.004
C01384=1143.398,101.048,-54.689,-179.248,6.664,149.003
C01385=1143.393,101.297,-54.709,-179.246,6.664,149.003
C01386=1143.388,101.546,-54.727,-179.243,6.666,149.003
C01387=1143.384,101.796,-54.745,-179.240,6.667,149.002
C01388=1143.379,102.045,-54.763,-179.237,6.669,149.001
C01389=1143.374,102.295,-54.781,-179.235,6.671,149.001
C01390=1143.369,102.543,-54.800,-179.232,6.672,149.001
C01391=1143.364,102.793,-54.818,-179.229,6.674,149.000
C01392=1143.359,103.042,-54.837,-179.226,6.676,149.000
C01393=1143.354,103.292,-54.854,-179.223,6.677,148.999
C01394=1143.349,103.541,-54.873,-179.220,6.679,148.999
C01395=1143.344,103.790,-54.892,-179.218,6.680,148.998
C01396=1143.340,104.040,-54.910,-179.216,6.681,148.998
C01397=1143.335,104.289,-54.928,-179.213,6.683,148.998
C01398=1143.330,104.538,-54.947,-179.210,6.685,148.997
C01399=1143.325,104.787,-54.966,-179.207,6.686,148.997
C01400=1143.320,105.037,-54.984,-179.204,6.688,148.996
C01401=1143.315,105.305,-55.004,-179.201,6.689,148.996
C01402=1143.310,105.573,-55.024,-179.199,6.691,148.995
C01403=1143.304,105.841,-55.044,-179.196,6.693,148.995
C01404=1143.300,106.110,-55.064,-179.192,6.695,148.994
C01405=1143.295,106.359,-55.082,-179.190,6.696,148.994
C01406=1143.289,106.608,-55.101,-179.187,6.698,148.993
C01407=1143.285,106.858,-55.119,-179.185,6.699,148.993
C01408=1143.280,107.107,-55.139,-179.182,6.701,148.993
C01409=1143.275,107.356,-55.156,-179.179,6.703,148.992
C01410=1143.271,107.606,-55.176,-179.176,6.704,148.992
C01411=1143.265,107.855,-55.194,-179.173,6.706,148.991
C01412=1143.260,108.104,-55.213,-179.170,6.707,148.991
C01413=1143.256,108.353,-55.231,-179.168,6.709,148.990
C01414=1143.251,108.602,-55.250,-179.165,6.711,148.990
C01415=1143.246,108.852,-55.268,-179.162,6.712,148.989
C01416=1143.241,109.101,-55.288,-179.160,6.714,148.989
C01417=1143.236,109.350,-55.306,-179.157,6.716,148.989
C01418=1143.232,109.600,-55.325,-179.154,6.717,148.988
C01419=1143.227,109.849,-55.344,-179.151,6.719,148.988
C01420=1143.222,110.098,-55.362,-179.149,6.720,148.987
C01421=1143.217,110.348,-55.381,-179.146,6.721,148.987
C01422=1143.212,110.596,-55.400,-179.143,6.723,148.986
C01423=1143.207,110.846,-55.419,-179.141,6.725,148.986
C01424=1143.203,111.095,-55.438,-179.138,6.726,148.986
C01425=1143.197,111.344,-55.457,-179.135,6.728,148.985
C01426=1143.193,111.594,-55.475,-179.132,6.730,148.985
C01427=1143.188,111.843,-55.495,-179.129,6.731,148.984
C01428=1143.183,112.093,-55.513,-179.126,6.733,148.984
C01429=1143.178,112.341,-55.532,-179.124,6.734,148.983
C01430=1143.173,112.590,-55.551,-179.121,6.736,148.983
C01431=1143.168,112.840,-55.570,-179.118,6.738,148.982
C01432=1143.164,113.089,-55.589,-179.116,6.739,148.982
C01433=1143.159,113.338,-55.608,-179.113,6.741,148.982
C01434=1143.154,113.587,-55.626,-179.110,6.743,148.981
C01435=1143.149,113.837,-55.646,-179.107,6.745,148.981
C01436=1143.144,114.086,-55.665,-179.105,6.746,148.980
C01437=1143.139,114.334,-55.684,-179.101,6.748,148.980
C01438=1143.134,114.585,-55.703,-179.099,6.749,148.979
C01439=1143.130,114.833,-55.721,-179.096,6.751,148.979
C01440=1143.125,115.083,-55.741,-179.093,6.753,148.979
C01441=1143.120,115.331,-55.760,-179.091,6.754,148.978
C01442=1143.115,115.581,-55.779,-179.088,6.756,148.978
C01443=1143.110,115.830,-55.798,-179.085,6.758,148.977
C01444=1143.106,116.080,-55.817,-179.082,6.759,148.977
C01445=1143.101,116.328,-55.836,-179.080,6.761,148.977
C01446=1143.096,116.578,-55.856,-179.077,6.763,148.976
C01447=1143.091,116.827,-55.874,-179.074,6.764,148.976
C01448=1143.086,117.077,-55.894,-179.071,6.766,148.975
C01449=1143.081,117.326,-55.913,-179.068,6.767,148.975
C01450=1143.077,117.575,-55.932,-179.066,6.769,148.974
C01451=1143.072,117.824,-55.952,-179.063,6.771,148.974
C01452=1143.067,118.073,-55.971,-179.060,6.773,148.974
C01453=1143.063,118.323,-55.990,-179.057,6.774,148.973
C01454=1143.057,118.571,-56.009,-179.055,6.776,148.973
C01455=1143.052,118.822,-56.028,-179.052,6.778,148.972
C01456=1143.048,119.070,-56.047,-179.049,6.779,148.972
C01457=1143.043,119.320,-56.067,-179.046,6.781,148.972
C01458=1143.038,119.569,-56.086,-179.044,6.783,148.971
C01459=1143.033,119.818,-56.106,-179.041,6.784,148.971
C01460=1143.029,120.067,-56.125,-179.038,6.786,148.970
C01461=1143.024,120.316,-56.144,-179.036,6.788,148.970
C01462=1143.019,120.566,-56.164,-179.033,6.789,148.969
C01463=1143.014,120.815,-56.183,-179.030,6.791,148.969
C01464=1143.010,121.064,-56.202,-179.027,6.793,148.969
C01465=1143.005,121.314,-56.222,-179.025,6.795,148.968
C01466=1142.999,121.562,-56.241,-179.021,6.796,148.968
C01467=1142.995,121.812,-56.261,-179.019,6.798,148.967
C01468=1142.990,122.060,-56.281,-179.016,6.799,148.967
C01469=1142.986,122.310,-56.300,-179.013,6.801,148.966
C01470=1142.981,122.559,-56.319,-179.011,6.803,148.966
C01471=1142.976,122.808,-56.339,-179.008,6.804,148.966
C01472=1142.971,123.058,-56.358,-179.005,6.806,148.965
C01473=1142.966,123.307,-56.378,-179.002,6.808,148.965
C01474=1142.961,123.556,-56.397,-178.999,6.810,148.964
C01475=1142.957,123.805,-56.416,-178.996,6.812,148.964
C01476=1142.952,124.054,-56.437,-178.994,6.814,148.964
C01477=1142.947,124.303,-56.456,-178.991,6.815,148.963
C01478=1142.942,124.553,-56.476,-178.988,6.817,148.963
C01479=1142.937,124.802,-56.495,-178.985,6.819,148.962
C01480=1142.932,125.051,-56.515,-178.983,6.820,148.962
C01481=1142.928,125.300,-56.535,-178.980,6.822,148.962
C01482=1142.923,125.550,-56.555,-178.977,6.824,148.961
C01483=1142.918,125.798,-56.573,-178.975,6.826,148.961
C01484=1142.914,126.048,-56.593,-178.972,6.827,148.960
C01485=1142.909,126.297,-56.613,-178.969,6.829,148.960
C01486=1142.904,126.546,-56.633,-178.966,6.831,148.960
C01487=1142.899,126.795,-56.652,-178.964,6.832,148.959
C01488=1142.894,127.045,-56.672,-178.961,6.834,148.959
C01489=1142.890,127.294,-56.692,-178.958,6.837,148.958
C01490=1142.885,127.542,-56.712,-178.955,6.838,148.958
C01491=1142.880,127.792,-56.731,-178.952,6.840,148.958
C01492=1142.875,128.041,-56.752,-178.949,6.842,148.957
C01493=1142.871,128.291,-56.771,-178.947,6.843,148.957
C01494=1142.865,128.539,-56.791,-178.944,6.845,148.956
C01495=1142.861,128.788,-56.811,-178.941,6.847,148.956
C01496=1142.856,129.038,-56.831,-178.939,6.848,148.956
C01497=1142.852,129.287,-56.851,-178.936,6.850,148.955
C01498=1142.846,129.536,-56.870,-178.933,6.852,148.955
C01499=1142.842,129.785,-56.890,-178.930,6.853,148.955
C01500=1142.837,130.034,-56.910,-178.927,6.856,148.954
C01501=1142.832,130.284,-56.930,-178.924,6.858,148.954
C01502=1142.827,130.532,-56.950,-178.922,6.859,148.953
C01503=1142.823,130.782,-56.970,-178.919,6.861,148.953
C01504=1142.817,131.031,-56.991,-178.916,6.863,148.953
C01505=1142.813,131.300,-57.012,-178.914,6.864,148.952
C01506=1142.808,131.568,-57.033,-178.910,6.867,148.952
C01507=1142.802,131.837,-57.055,-178.907,6.868,148.951
C01508=1142.797,132.105,-57.076,-178.904,6.870,148.951
C01509=1142.793,132.355,-57.096,-178.901,6.873,148.950
C01510=1142.787,132.604,-57.117,-178.898,6.874,148.950
C01511=1142.782,132.852,-57.137,-178.896,6.876,148.950
C01512=1142.778,133.102,-57.156,-178.893,6.878,148.949
C01513=1142.773,133.351,-57.177,-178.890,6.879,148.949
C01514=1142.768,133.600,-57.196,-178.887,6.881,148.948
C01515=1142.764,133.849,-57.217,-178.885,6.883,148.948
C01516=1142.759,134.099,-57.238,-178.882,6.884,148.948
C01517=1142.754,134.347,-57.257,-178.879,6.887,148.947
C01518=1142.749,134.596,-57.277,-178.876,6.889,148.947
C01519=1142.744,134.846,-57.297,-178.874,6.891,148.947
C01520=1142.740,135.095,-57.318,-178.871,6.892,148.946
C01521=1142.735,135.344,-57.338,-178.868,6.894,148.946
C01522=1142.730,135.593,-57.359,-178.866,6.896,148.945
C01523=1142.726,135.843,-57.379,-178.863,6.898,148.945
C01524=1142.721,136.092,-57.399,-178.860,6.900,148.945
C01525=1142.717,136.341,-57.419,-178.857,6.902,148.944
C01526=1142.711,136.590,-57.439,-178.854,6.903,148.944
C01527=1142.706,136.839,-57.460,-178.851,6.905,148.944
C01528=1142.702,137.088,-57.480,-178.849,6.907,148.943
C01529=1142.697,137.337,-57.501,-178.846,6.909,148.943
C01530=1142.692,137.587,-57.521,-178.843,6.911,148.942
C01531=1142.687,137.835,-57.541,-178.840,6.913,148.942
C01532=1142.683,138.084,-57.561,-178.837,6.915,148.942
C01533=1142.678,138.334,-57.582,-178.834,6.916,148.941
C01534=1142.673,138.583,-57.603,-178.832,6.918,148.941
C01535=1142.669,138.832,-57.622,-178.829,6.920,148.940
C01536=1142.663,139.081,-57.643,-178.826,6.922,148.940
C01537=1142.659,139.330,-57.664,-178.823,6.924,148.940
C01538=1142.655,139.579,-57.684,-178.821,6.926,148.939
C01539=1142.649,139.829,-57.705,-178.818,6.928,148.939
C01540=1142.645,140.078,-57.725,-178.815,6.929,148.939
C01541=1142.640,140.326,-57.746,-178.813,6.931,148.938
C01542=1142.635,140.576,-57.767,-178.809,6.934,148.938
C01543=1142.631,140.825,-57.787,-178.807,6.935,148.938
C01544=1142.626,141.074,-57.808,-178.804,6.937,148.937
C01545=1142.621,141.324,-57.828,-178.801,6.939,148.937
C01546=1142.617,141.572,-57.848,-178.798,6.940,148.936
C01547=1142.611,141.822,-57.869,-178.795,6.943,148.936
C01548=1142.607,142.071,-57.889,-178.792,6.945,148.936
C01549=1142.602,142.320,-57.910,-178.790,6.946,148.935
C01550=1142.597,142.569,-57.931,-178.787,6.948,148.935
C01551=1142.593,142.818,-57.951,-178.785,6.950,148.935
C01552=1142.588,143.067,-57.972,-178.781,6.953,148.934
C01553=1142.584,143.315,-57.993,-178.779,6.954,148.934
C01554=1142.578,143.565,-58.014,-178.776,6.956,148.934
C01555=1142.574,143.814,-58.034,-178.773,6.958,148.933
C01556=1142.569,144.063,-58.055,-178.771,6.959,148.933
C01557=1142.564,144.312,-58.076,-178.767,6.962,148.932
C01558=1142.559,144.561,-58.097,-178.765,6.964,148.932
C01559=1142.555,144.810,-58.117,-178.762,6.965,148.932
C01560=1142.550,145.059,-58.138,-178.759,6.967,148.931
C01561=1142.546,145.309,-58.159,-178.757,6.969,148.931
C01562=1142.541,145.558,-58.180,-178.754,6.972,148.931
C01563=1142.536,145.807,-58.201,-178.751,6.973,148.930
C01564=1142.531,146.056,-58.222,-178.748,6.975,148.930
C01565=1142.526,146.305,-58.243,-178.745,6.977,148.930
C01566=1142.522,146.554,-58.263,-178.742,6.979,148.929
C01567=1142.516,146.803,-58.284,-178.739,6.981,148.929
C01568=1142.512,147.052,-58.305,-178.737,6.983,148.928
C01569=1142.507,147.301,-58.326,-178.735,6.985,148.928
C01570=1142.503,147.551,-58.347,-178.731,6.987,148.928
C01571=1142.498,147.800,-58.368,-178.729,6.989,148.927
C01572=1142.493,148.048,-58.390,-178.726,6.991,148.927
C01573=1142.489,148.297,-58.410,-178.723,6.992,148.927
C01574=1142.484,148.547,-58.431,-178.720,6.995,148.926
C01575=1142.478,148.796,-58.452,-178.717,6.997,148.926
C01576=1142.474,149.044,-58.473,-178.714,6.998,148.926
C01577=1142.470,149.294,-58.494,-178.712,7.000,148.925
C01578=1142.465,149.543,-58.515,-178.709,7.003,148.925
C01579=1142.460,149.792,-58.536,-178.706,7.005,148.925
C01580=1142.455,150.041,-58.557,-178.703,7.006,148.924
C01581=1142.450,150.290,-58.578,-178.701,7.008,148.924
C01582=1142.446,150.539,-58.599,-178.697,7.011,148.923
C01583=1142.441,150.789,-58.621,-178.695,7.012,148.923
C01584=1142.437,151.037,-58.642,-178.692,7.014,148.923
C01585=1142.432,151.286,-58.663,-178.690,7.016,148.923
C01586=1142.427,151.535,-58.684,-178.686,7.019,148.922
C01587=1142.422,151.784,-58.705,-178.684,7.020,148.922
C01588=1142.417,152.034,-58.727,-178.681,7.022,148.921
C01589=1142.413,152.282,-58.748,-178.678,7.024,148.921
C01590=1142.408,152.532,-58.769,-178.675,7.027,148.921
C01591=1142.403,152.780,-58.790,-178.673,7.028,148.921
C01592=1142.399,153.030,-58.812,-178.670,7.030,148.920
C01593=1142.395,153.279,-58.833,-178.667,7.033,148.920
C01594=1142.389,153.528,-58.854,-178.664,7.034,148.919
C01595=1142.385,153.776,-58.876,-178.661,7.036,148.919
C01596=1142.380,154.026,-58.897,-178.659,7.038,148.919
C01597=1142.375,154.275,-58.919,-178.656,7.041,148.918
C01598=1142.370,154.524,-58.940,-178.653,7.042,148.918
C01599=1142.366,154.773,-58.961,-178.650,7.044,148.918
C01600=1142.362,155.022,-58.983,-178.647,7.047,148.917
C01601=1142.356,155.271,-59.004,-178.645,7.049,148.917
C01602=1142.351,155.520,-59.025,-178.642,7.050,148.917
C01603=1142.347,155.769,-59.047,-178.639,7.053,148.916
C01604=1142.342,156.018,-59.068,-178.636,7.055,148.916
C01605=1142.337,156.267,-59.090,-178.633,7.056,148.916
C01606=1142.334,156.516,-59.111,-178.631,7.058,148.915
C01607=1142.328,156.765,-59.132,-178.628,7.061,148.915
C01608=1142.324,157.014,-59.154,-178.625,7.063,148.915
C01609=1142.318,157.283,-59.177,-178.622,7.065,148.914
C01610=1142.314,157.552,-59.201,-178.619,7.067,148.914
C01611=1142.308,157.821,-59.224,-178.616,7.069,148.914
C01612=1142.303,158.090,-59.247,-178.613,7.071,148.913
C01613=1142.299,158.339,-59.269,-178.610,7.074,148.913
C01614=1142.294,158.588,-59.291,-178.608,7.076,148.913
C01615=1142.289,158.837,-59.313,-178.605,7.077,148.912
C01616=1142.284,159.086,-59.333,-178.602,7.080,148.912
C01617=1142.280,159.335,-59.356,-178.599,7.082,148.912
C01618=1142.275,159.584,-59.377,-178.596,7.083,148.911
C01619=1142.271,159.833,-59.399,-178.593,7.086,148.911
C01620=1142.266,160.082,-59.421,-178.591,7.088,148.911
C01621=1142.261,160.331,-59.442,-178.588,7.090,148.910
C01622=1142.257,160.581,-59.464,-178.585,7.092,148.910
C01623=1142.252,160.829,-59.486,-178.582,7.094,148.910
C01624=1142.247,161.079,-59.508,-178.580,7.096,148.910
C01625=1142.243,161.327,-59.529,-178.576,7.099,148.909
C01626=1142.238,161.576,-59.551,-178.574,7.100,148.909
C01627=1142.233,161.825,-59.573,-178.570,7.103,148.908
C01628=1142.229,162.074,-59.595,-178.568,7.105,148.908
C01629=1142.224,162.323,-59.617,-178.566,7.107,148.908
C01630=1142.219,162.572,-59.639,-178.562,7.109,148.908
C01631=1142.214,162.822,-59.661,-178.560,7.111,148.907
C01632=1142.210,163.070,-59.683,-178.557,7.113,148.907
C01633=1142.205,163.319,-59.705,-178.554,7.116,148.907
C01634=1142.200,163.568,-59.727,-178.551,7.117,148.906
C01635=1142.196,163.817,-59.748,-178.549,7.119,148.906
C01636=1142.191,164.066,-59.770,-178.546,7.122,148.906
C01637=1142.186,164.315,-59.792,-178.543,7.124,148.905
C01638=1142.182,164.564,-59.814,-178.540,7.126,148.905
C01639=1142.177,164.813,-59.836,-178.537,7.128,148.905
C01640=1142.172,165.062,-59.858,-178.535,7.130,148.904
C01641=1142.167,165.311,-59.880,-178.532,7.132,148.904
C01642=1142.163,165.560,-59.902,-178.529,7.134,148.904
C01643=1142.158,165.809,-59.924,-178.527,7.136,148.904
C01644=1142.154,166.058,-59.946,-178.523,7.139,148.903
C01645=1142.148,166.307,-59.968,-178.521,7.140,148.903
C01646=1142.144,166.556,-59.991,-178.517,7.143,148.903
C01647=1142.140,166.805,-60.013,-178.515,7.145,148.902
C01648=1142.135,167.054,-60.035,-178.512,7.147,148.902
C01649=1142.130,167.303,-60.056,-178.509,7.149,148.902
C01650=1142.125,167.552,-60.079,-178.506,7.151,148.901
C01651=1142.121,167.801,-60.102,-178.504,7.154,148.901
C01652=1142.117,168.050,-60.123,-178.501,7.156,148.901
C01653=1142.112,168.299,-60.145,-178.498,7.157,148.900
C01654=1142.107,168.548,-60.168,-178.495,7.160,148.900
C01655=1142.102,168.797,-60.190,-178.493,7.162,148.900
C01656=1142.098,169.045,-60.212,-178.489,7.165,148.900
C01657=1142.093,169.295,-60.235,-178.487,7.167,148.899
C01658=1142.088,169.544,-60.256,-178.484,7.168,148.899
C01659=1142.084,169.792,-60.279,-178.481,7.171,148.899
C01660=1142.079,170.042,-60.302,-178.478,7.173,148.898
C01661=1142.074,170.291,-60.324,-178.476,7.175,148.898
C01662=1142.070,170.539,-60.346,-178.473,7.177,148.898
C01663=1142.065,170.788,-60.369,-178.470,7.179,148.897
C01664=1142.060,171.038,-60.391,-178.467,7.182,148.897
C01665=1142.056,171.286,-60.413,-178.465,7.184,148.897
C01666=1142.051,171.535,-60.436,-178.461,7.186,148.897
C01667=1142.047,171.784,-60.458,-178.459,7.188,148.896
C01668=1142.042,172.034,-60.481,-178.456,7.191,148.896
C01669=1142.037,172.282,-60.503,-178.453,7.192,148.896
C01670=1142.033,172.531,-60.526,-178.450,7.195,148.896
C01671=1142.028,172.781,-60.548,-178.448,7.197,148.895
C01672=1142.023,173.029,-60.571,-178.445,7.199,148.895
C01673=1142.018,173.278,-60.593,-178.442,7.202,148.895
C01674=1142.014,173.526,-60.616,-178.439,7.203,148.894
C01675=1142.010,173.776,-60.638,-178.436,7.206,148.894
C01676=1142.005,174.025,-60.661,-178.434,7.208,148.894
C01677=1142.001,174.274,-60.683,-178.431,7.211,148.893
C01678=1141.995,174.522,-60.706,-178.428,7.212,148.893
C01679=1141.991,174.772,-60.728,-178.425,7.215,148.893
C01680=1141.986,175.021,-60.751,-178.422,7.217,148.893
C01681=1141.981,175.269,-60.773,-178.420,7.219,148.892
C01682=1141.977,175.519,-60.797,-178.417,7.222,148.892
C01683=1141.973,175.767,-60.819,-178.414,7.223,148.892
C01684=1141.967,176.016,-60.842,-178.411,7.226,148.891
C01685=1141.963,176.265,-60.864,-178.409,7.228,148.891
C01686=1141.958,176.514,-60.888,-178.405,7.230,148.891
C01687=1141.954,176.763,-60.910,-178.403,7.232,148.891
C01688=1141.949,177.012,-60.933,-178.400,7.235,148.890
C01689=1141.944,177.261,-60.956,-178.397,7.237,148.890
C01690=1141.940,177.510,-60.978,-178.394,7.240,148.890
C01691=1141.935,177.759,-61.001,-178.392,7.241,148.890
C01692=1141.931,178.007,-61.024,-178.388,7.244,148.889
C01693=1141.926,178.257,-61.047,-178.386,7.246,148.889
C01694=1141.922,178.505,-61.069,-178.383,7.249,148.889
C01695=1141.917,178.754,-61.093,-178.380,7.250,148.888
C01696=1141.912,179.003,-61.116,-178.377,7.253,148.888
C01697=1141.907,179.252,-61.138,-178.375,7.255,148.888
C01698=1141.903,179.501,-61.161,-178.372,7.258,148.888
C01699=1141.898,179.750,-61.184,-178.369,7.260,148.887
C01700=1141.894,179.999,-61.207,-178.366,7.262,148.887
C01701=1141.889,180.248,-61.231,-178.364,7.264,148.887
C01702=1141.885,180.497,-61.252,-178.360,7.267,148.887
C01703=1141.880,180.746,-61.276,-178.358,7.269,148.886
C01704=1141.875,180.995,-61.299,-178.355,7.271,148.886
C01705=1141.870,181.244,-61.322,-178.352,7.273,148.886
C01706=1141.866,181.492,-61.345,-178.349,7.276,148.886
C01707=1141.862,181.741,-61.368,-178.347,7.278,148.885
C01708=1141.856,181.990,-61.391,-178.344,7.281,148.885
C01709=1141.852,182.238,-61.414,-178.341,7.282,148.885
C01710=1141.848,182.488,-61.438,-178.338,7.285,148.884
C01711=1141.843,182.737,-61.461,-178.336,7.287,148.884
C01712=1141.838,182.986,-61.484,-178.332,7.289,148.884
C01713=1141.834,183.255,-61.509,-178.330,7.292,148.884
C01714=1141.828,183.525,-61.534,-178.327,7.294,148.883
C01715=1141.823,183.795,-61.559,-178.323,7.297,148.883
C01716=1141.818,184.064,-61.584,-178.320,7.299,148.883
C01717=1141.814,184.313,-61.607,-178.318,7.301,148.883
C01718=1141.809,184.562,-61.630,-178.315,7.304,148.882
C01719=1141.805,184.810,-61.654,-178.312,7.307,148.882
C01720=1141.800,185.060,-61.677,-178.309,7.308,148.882
C01721=1141.795,185.309,-61.701,-178.306,7.311,148.882
C01722=1141.791,185.557,-61.723,-178.304,7.313,148.881
C01723=1141.787,185.806,-61.747,-178.300,7.316,148.881
C01724=1141.782,186.055,-61.770,-178.298,7.318,148.881
C01725=1141.777,186.304,-61.794,-178.295,7.320,148.880
C01726=1141.773,186.553,-61.817,-178.293,7.322,148.880
C01727=1141.768,186.802,-61.840,-178.289,7.325,148.880
C01728=1141.763,187.050,-61.864,-178.287,7.327,148.880
C01729=1141.758,187.299,-61.887,-178.284,7.329,148.880
C01730=1141.754,187.548,-61.910,-178.281,7.332,148.879
C01731=1141.750,187.797,-61.933,-178.278,7.334,148.879
C01732=1141.745,188.046,-61.957,-178.276,7.337,148.879
C01733=1141.740,188.294,-61.981,-178.273,7.339,148.879
C01734=1141.736,188.543,-62.004,-178.270,7.342,148.878
C01735=1141.731,188.792,-62.028,-178.267,7.343,148.878
C01736=1141.726,189.041,-62.051,-178.264,7.346,148.878
C01737=1141.722,189.290,-62.075,-178.262,7.348,148.878
C01738=1141.717,189.539,-62.098,-178.259,7.351,148.877
C01739=1141.713,189.788,-62.122,-178.256,7.353,148.877
C01740=1141.708,190.037,-62.145,-178.253,7.355,148.877
C01741=1141.704,190.285,-62.169,-178.250,7.358,148.877
C01742=1141.699,190.534,-62.193,-178.248,7.360,148.876
C01743=1141.694,190.783,-62.216,-178.245,7.363,148.876
C01744=1141.690,191.032,-62.240,-178.241,7.365,148.876
C01745=1141.685,191.281,-62.263,-178.239,7.367,148.876
C01746=1141.681,191.529,-62.287,-178.236,7.370,148.875
C01747=1141.676,191.778,-62.311,-178.234,7.372,148.875
C01748=1141.672,192.028,-62.334,-178.230,7.375,148.875
C01749=1141.667,192.277,-62.359,-178.228,7.377,148.875
C01750=1141.663,192.526,-62.382,-178.225,7.379,148.874
C01751=1141.658,192.774,-62.406,-178.222,7.382,148.874
C01752=1141.653,193.023,-62.430,-178.219,7.384,148.874
C01753=1141.648,193.272,-62.454,-178.217,7.387,148.874
C01754=1141.644,193.521,-62.477,-178.214,7.388,148.874
C01755=1141.639,193.769,-62.501,-178.211,7.391,148.873
C01756=1141.635,194.018,-62.525,-178.208,7.394,148.873
C01757=1141.630,194.267,-62.549,-178.206,7.396,148.873
C01758=1141.626,194.516,-62.572,-178.203,7.399,148.873
C01759=1141.621,194.764,-62.596,-178.200,7.401,148.872
C01760=1141.616,195.014,-62.621,-178.197,7.404,148.872
C01761=1141.612,195.263,-62.645,-178.194,7.406,148.872
C01762=1141.607,195.512,-62.668,-178.192,7.408,148.872
C01763=1141.603,195.760,-62.692,-178.189,7.411,148.872
C01764=1141.598,196.008,-62.716,-178.186,7.414,148.871
C01765=1141.594,196.257,-62.740,-178.183,7.415,148.871
C01766=1141.589,196.506,-62.764,-178.180,7.418,148.871
C01767=1141.585,196.755,-62.789,-178.177,7.421,148.871
C01768=1141.580,197.004,-62.812,-178.175,7.423,148.870
C01769=1141.576,197.253,-62.836,-178.172,7.426,148.870
C01770=1141.571,197.501,-62.861,-178.169,7.428,148.870
C01771=1141.566,197.750,-62.884,-178.166,7.430,148.870
C01772=1141.562,197.999,-62.908,-178.163,7.433,148.870
C01773=1141.558,198.248,-62.933,-178.161,7.435,148.869
C01774=1141.553,198.497,-62.957,-178.158,7.438,148.869
C01775=1141.548,198.746,-62.981,-178.155,7.441,148.869
C01776=1141.544,198.994,-63.005,-178.152,7.442,148.869
C01777=1141.539,199.243,-63.029,-178.149,7.445,148.869
C01778=1141.535,199.492,-63.054,-178.147,7.448,148.868
C01779=1141.530,199.741,-63.077,-178.144,7.450,148.868
C01780=1141.526,199.989,-63.101,-178.141,7.453,148.868
C01781=1141.520,200.238,-63.126,-178.138,7.455,148.868
C01782=1141.517,200.487,-63.150,-178.136,7.457,148.868
C01783=1141.512,200.736,-63.175,-178.133,7.460,148.867
C01784=1141.507,200.984,-63.199,-178.129,7.463,148.867
C01785=1141.503,201.233,-63.223,-178.127,7.465,148.867
C01786=1141.499,201.482,-63.248,-178.124,7.467,148.867
C01787=1141.493,201.731,-63.272,-178.121,7.470,148.867
C01788=1141.489,201.980,-63.296,-178.119,7.472,148.866
C01789=1141.484,202.228,-63.320,-178.116,7.475,148.866
C01790=1141.480,202.478,-63.345,-178.113,7.478,148.866
C01791=1141.476,202.726,-63.369,-178.110,7.480,148.866
C01792=1141.471,202.975,-63.394,-178.107,7.483,148.865
C01793=1141.467,203.224,-63.418,-178.105,7.485,148.865
C01794=1141.462,203.472,-63.443,-178.102,7.487,148.865
C01795=1141.457,203.721,-63.467,-178.099,7.490,148.865
C01796=1141.453,203.970,-63.492,-178.096,7.493,148.865
C01797=1141.448,204.219,-63.516,-178.094,7.495,148.864
C01798=1141.444,204.467,-63.540,-178.091,7.498,148.864
C01799=1141.439,204.717,-63.565,-178.087,7.500,148.864
C01800=1141.435,204.965,-63.589,-178.085,7.502,148.864
C01801=1141.430,205.213,-63.614,-178.082,7.505,148.864
C01802=1141.426,205.463,-63.639,-178.079,7.508,148.863
C01803=1141.421,205.711,-63.664,-178.076,7.511,148.863
C01804=1141.416,205.960,-63.688,-178.074,7.512,148.863
C01805=1141.412,206.209,-63.713,-178.071,7.515,148.863
C01806=1141.407,206.457,-63.737,-178.068,7.518,148.863
C01807=1141.403,206.706,-63.761,-178.065,7.520,148.862
C01808=1141.398,206.955,-63.786,-178.063,7.523,148.862
C01809=1141.394,207.203,-63.811,-178.060,7.526,148.862
C01810=1141.389,207.452,-63.836,-178.057,7.527,148.862
C01811=1141.385,207.701,-63.861,-178.054,7.530,148.862
C01812=1141.380,207.950,-63.885,-178.051,7.533,148.862
C01813=1141.376,208.198,-63.911,-178.048,7.536,148.861
C01814=1141.372,208.447,-63.935,-178.046,7.538,148.861
C01815=1141.366,208.696,-63.959,-178.043,7.541,148.861
C01816=1141.362,208.945,-63.985,-178.040,7.543,148.861
C01817=1141.357,209.215,-64.011,-178.037,7.546,148.861
C01818=1141.352,209.486,-64.038,-178.034,7.549,148.860
C01819=1141.348,209.757,-64.065,-178.031,7.552,148.860
C01820=1141.342,210.027,-64.092,-178.028,7.555,148.860
C01821=1141.338,210.276,-64.118,-178.025,7.557,148.860
C01822=1141.333,210.525,-64.143,-178.022,7.560,148.860
C01823=1141.330,210.773,-64.168,-178.020,7.562,148.860
C01824=1141.324,211.022,-64.192,-178.017,7.565,148.859
C01825=1141.319,211.271,-64.217,-178.014,7.568,148.859
C01826=1141.316,211.519,-64.242,-178.011,7.571,148.859
C01827=1141.311,211.768,-64.267,-178.008,7.572,148.859
C01828=1141.307,212.017,-64.293,-178.006,7.575,148.859
C01829=1141.301,212.265,-64.317,-178.003,7.578,148.859
C01830=1141.298,212.514,-64.342,-178.000,7.581,148.859
C01831=1141.293,212.763,-64.367,-177.997,7.583,148.858
C01832=1141.289,213.011,-64.393,-177.994,7.586,148.858
C01833=1141.283,213.260,-64.418,-177.992,7.589,148.858
C01834=1141.280,213.509,-64.443,-177.988,7.591,148.858
